KUKA KRL program: MyProgram_230().src

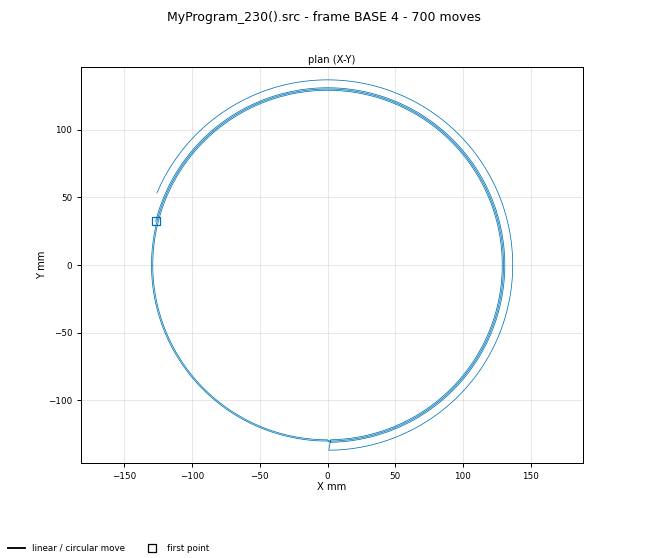
[picture p0: tool path of MyProgram_230().src in frame BASE 4, 700 of 700 moves have a stored position in this frame; points joined in program order, loops and branches not executed]
&ACCESS RVP
&REL 1
&PARAM TEMPLATE = C:\KRC\Roboter\Template\vorgabe
&PARAM EDITMASK = *
DEF MyProgram_230()
; ---- Setting reference (Base) ----
$BASE = BASE_DATA[4]

; --------------------------
; ---- Setting tool (TCP) ----
$TOOL = TOOL_DATA[3]
; --------------------------

$VEL.CP = VEL_APROX_PRINT
Startdeposition()
$VEL.CP = VEL_PRINT
LIN {X -126.9294,Y 32.2253,Z 157,A 163.8285,B 18.3414,C -0.4875,E1 18.1927,E2 284.7259} C_DIS
LIN {X -125.904,Y 36.0324,Z 157,A 161.9446,B 18.3414,C -0.4875,E1 18.1941,E2 286.6256} C_DIS
LIN {X -124.7405,Y 39.8661,Z 157,A 160.3345,B 18.3411,C -0.4975,E1 18.1954,E2 288.2164} C_DIS
LIN {X -123.6623,Y 43.0949,Z 157,A 158.8283,B 18.3411,C -0.5013,E1 18.1968,E2 289.7223} C_DIS
LIN {X -122.5468,Y 46.1718,Z 157,A 157.3766,B 18.3409,C -0.5049,E1 18.1982,E2 291.1743} C_DIS
LIN {X -121.4032,Y 49.0996,Z 157,A 155.9825,B 18.3409,C -0.5083,E1 18.1996,E2 292.5684} C_DIS
LIN {X -119.9916,Y 52.4573,Z 157,A 154.3901,B 18.3407,C -0.513,E1 18.2013,E2 294.1583} C_DIS
LIN {X -117.3041,Y 58.2179,Z 157,A 151.6663,B 18.3405,C -0.5228,E1 18.2046,E2 296.8714} C_DIS
LIN {X -116.1041,Y 60.5758,Z 157,A 149.9342,B 18.3409,C -0.5068,E1 18.2069,E2 298.6678} C_DIS
LIN {X -114.0894,Y 64.2932,Z 157,A 148.54,B 18.3403,C -0.5272,E1 18.2087,E2 300.007} C_DIS
LIN {X -112.0031,Y 67.8624,Z 157,A 146.6599,B 18.3403,C -0.5297,E1 18.2114,E2 301.8927} C_DIS
LIN {X -109.7276,Y 71.4835,Z 157,A 144.7555,B 18.3402,C -0.5336,E1 18.2143,E2 303.7982} C_DIS
LIN {X -107.2573,Y 75.1401,Z 157,A 142.8027,B 18.34,C -0.5379,E1 18.2174,E2 305.7508} C_DIS
LIN {X -104.7432,Y 78.6064,Z 157,A 140.9069,B 18.34,C -0.542,E1 18.2205,E2 307.6465} C_DIS
LIN {X -102.0917,Y 82.0203,Z 157,A 138.9861,B 18.3398,C -0.5458,E1 18.2238,E2 309.568} C_DIS
LIN {X -99.1429,Y 85.561,Z 157,A 136.9936,B 18.3396,C -0.5515,E1 18.2274,E2 311.5549} C_DIS
LIN {X -96.2928,Y 88.7565,Z 157,A 135.0913,B 18.3396,C -0.555,E1 18.231,E2 313.4579} C_DIS
LIN {X -93.2172,Y 91.982,Z 157,A 133.0947,B 18.3395,C -0.5579,E1 18.2349,E2 315.4573} C_DIS
LIN {X -90.087,Y 95.0495,Z 157,A 131.1811,B 18.3393,C -0.5624,E1 18.2387,E2 317.3678} C_DIS
LIN {X -86.7985,Y 98.0612,Z 157,A 129.232,B 18.3392,C -0.5667,E1 18.2428,E2 319.3141} C_DIS
LIN {X -83.2978,Y 101.0522,Z 157,A 127.211,B 18.3391,C -0.5707,E1 18.2471,E2 321.3333} C_DIS
LIN {X -79.8786,Y 103.7765,Z 157,A 125.2544,B 18.3391,C -0.573,E1 18.2514,E2 323.2926} C_DIS
LIN {X -76.3559,Y 106.3946,Z 157,A 123.3696,B 18.3389,C -0.5779,E1 18.2556,E2 325.1709} C_DIS
LIN {X -72.8799,Y 108.8051,Z 157,A 121.4838,B 18.3388,C -0.5802,E1 18.26,E2 327.0585} C_DIS
LIN {X -69.4414,Y 111.0314,Z 157,A 119.7018,B 18.3387,C -0.5837,E1 18.2642,E2 328.8372} C_DIS
LIN {X -65.8977,Y 113.1706,Z 157,A 117.8352,B 18.3387,C -0.5848,E1 18.2687,E2 330.7082} C_DIS
LIN {X -61.9917,Y 115.356,Z 157,A 115.6717,B 18.3387,C -0.5808,E1 18.274,E2 332.893} C_DIS
LIN {X -59.1213,Y 116.8514,Z 157,A 114.6066,B 18.3383,C -0.5952,E1 18.2766,E2 333.9162} C_DIS
LIN {X -56.0403,Y 118.3603,Z 157,A 112.9696,B 18.3384,C -0.5927,E1 18.2807,E2 335.5674} C_DIS
LIN {X -48.8655,Y 121.4976,Z 157,A 109.6259,B 18.3382,C -0.6001,E1 18.2893,E2 338.8981} C_DIS
LIN {X -45.691,Y 122.7269,Z 157,A 108.1493,B 18.3381,C -0.6024,E1 18.2931,E2 340.3718} C_DIS
LIN {X -42.2196,Y 123.9658,Z 157,A 106.4116,B 18.3381,C -0.5998,E1 18.2977,E2 342.1225} C_DIS
LIN {X -38.1423,Y 125.2785,Z 157,A 104.655,B 18.338,C -0.606,E1 18.3024,E2 343.8638} C_DIS
LIN {X -35.0335,Y 126.1834,Z 157,A 103.2075,B 18.338,C -0.6062,E1 18.3062,E2 345.3137} C_DIS
LIN {X -27.6513,Y 128.0037,Z 157,A 99.8455,B 18.338,C -0.6078,E1 18.3154,E2 348.6771} C_DIS
LIN {X -20.6201,Y 129.3241,Z 157,A 96.6623,B 18.338,C -0.6079,E1 18.3241,E2 351.8643} C_DIS
LIN {X -15.0154,Y 130.093,Z 157,A 94.0812,B 18.338,C -0.6054,E1 18.3313,E2 354.456} C_DIS
LIN {X -11.0032,Y 130.4934,Z 157,A 92.4941,B 18.3378,C -0.6126,E1 18.3357,E2 356.0216} C_DIS
LIN {X -6.9018,Y 130.7749,Z 157,A 90.6614,B 18.3378,C -0.6119,E1 18.3408,E2 357.8572} C_DIS
LIN {X -3.0947,Y 130.9211,Z 157,A 89.0121,B 18.3378,C -0.6129,E1 18.3454,E2 359.5036} C_DIS
LIN {X 0.7077,Y 130.9547,Z 157,A 87.3244,B 18.3378,C -0.6123,E1 18.3501,E2 361.1932} C_DIS
LIN {X 4.9525,Y 130.8629,Z 157,A 85.4948,B 18.3378,C -0.6134,E1 18.3552,E2 363.0188} C_DIS
LIN {X 8.8445,Y 130.6593,Z 157,A 83.69,B 18.3378,C -0.6096,E1 18.3603,E2 364.8345} C_DIS
LIN {X 12.681,Y 130.3411,Z 157,A 82.1185,B 18.3378,C -0.6135,E1 18.3646,E2 366.3922} C_DIS
LIN {X 16.8208,Y 129.8718,Z 157,A 80.0899,B 18.338,C -0.6055,E1 18.3703,E2 368.4441} C_DIS
LIN {X 21.4829,Y 129.1822,Z 157,A 78.2047,B 18.3378,C -0.6113,E1 18.3754,E2 370.3082} C_DIS
LIN {X 26.623,Y 128.2226,Z 157,A 75.8818,B 18.3378,C -0.6089,E1 18.3818,E2 372.6348} C_DIS
LIN {X 30.47,Y 127.3623,Z 157,A 74.2016,B 18.3378,C -0.6096,E1 18.3864,E2 374.3096} C_DIS
LIN {X 34.0088,Y 126.4635,Z 157,A 72.3281,B 18.3382,C -0.5982,E1 18.3915,E2 376.2149} C_DIS
LIN {X 37.1976,Y 125.5629,Z 157,A 71.2631,B 18.3378,C -0.6115,E1 18.3942,E2 377.2351} C_DIS
LIN {X 39.9846,Y 124.7027,Z 157,A 69.9298,B 18.3379,C -0.6084,E1 18.3978,E2 378.575} C_DIS
LIN {X 43.2512,Y 123.6082,Z 157,A 68.3028,B 18.3381,C -0.6025,E1 18.4021,E2 380.2161} C_DIS
LIN {X 47.2394,Y 122.1392,Z 157,A 66.5756,B 18.338,C -0.6057,E1 18.4066,E2 381.9279} C_DIS
LIN {X 50.5263,Y 120.8163,Z 157,A 64.9972,B 18.338,C -0.603,E1 18.4107,E2 383.5097} C_DIS
LIN {X 53.888,Y 119.3557,Z 157,A 63.2995,B 18.3383,C -0.5976,E1 18.4151,E2 385.2186} C_DIS
LIN {X 57.8507,Y 117.4852,Z 157,A 61.4569,B 18.3383,C -0.5981,E1 18.4197,E2 387.0529} C_DIS
LIN {X 60.9785,Y 115.8926,Z 157,A 59.9952,B 18.3383,C -0.599,E1 18.4233,E2 388.5062} C_DIS
LIN {X 64.5859,Y 113.9244,Z 157,A 58.0353,B 18.3385,C -0.5902,E1 18.4281,E2 390.4856} C_DIS
LIN {X 68.6354,Y 111.5312,Z 157,A 56.0373,B 18.3385,C -0.5895,E1 18.4329,E2 392.4773} C_DIS
LIN {X 72.3786,Y 109.1397,Z 157,A 54.0704,B 18.3386,C -0.5855,E1 18.4375,E2 394.4477} C_DIS
LIN {X 76.0983,Y 106.5788,Z 157,A 52.1676,B 18.3386,C -0.585,E1 18.4418,E2 396.3427} C_DIS
LIN {X 79.4898,Y 104.0738,Z 157,A 50.3093,B 18.3388,C -0.5813,E1 18.446,E2 398.2034} C_DIS
LIN {X 83.6518,Y 100.759,Z 157,A 47.9853,B 18.3388,C -0.5771,E1 18.451,E2 400.5282} C_DIS
LIN {X 87.0752,Y 97.8164,Z 157,A 45.6005,B 18.3395,C -0.5574,E1 18.4561,E2 402.962} C_DIS
LIN {X 90.2686,Y 94.877,Z 157,A 44.2587,B 18.3389,C -0.5752,E1 18.4587,E2 404.2399} C_DIS
LIN {X 92.9547,Y 92.2464,Z 157,A 42.5188,B 18.3392,C -0.5681,E1 18.4622,E2 405.992} C_DIS
LIN {X 96.4427,Y 88.5934,Z 157,A 40.3208,B 18.3392,C -0.5637,E1 18.4664,E2 408.1902} C_DIS
LIN {X 99.4064,Y 85.2551,Z 157,A 38.0738,B 18.3398,C -0.5478,E1 18.4706,E2 410.4732} C_DIS
LIN {X 101.7587,Y 82.4332,Z 157,A 36.8229,B 18.3395,C -0.5581,E1 18.4727,E2 411.6836} C_DIS
LIN {X 104.2925,Y 79.2036,Z 157,A 34.942,B 18.3397,C -0.5505,E1 18.4759,E2 413.5759} C_DIS
LIN {X 107.0744,Y 75.3993,Z 157,A 32.7589,B 18.34,C -0.5407,E1 18.4795,E2 415.775} C_DIS
LIN {X 109.5714,Y 71.7232,Z 157,A 31.0093,B 18.3399,C -0.5435,E1 18.4822,E2 417.5036} C_DIS
LIN {X 111.8857,Y 68.0565,Z 157,A 29.089,B 18.34,C -0.5377,E1 18.485,E2 419.4285} C_DIS
LIN {X 114.0229,Y 64.4115,Z 157,A 27.2622,B 18.3402,C -0.5338,E1 18.4876,E2 421.2545} C_DIS
LIN {X 116.1297,Y 60.5271,Z 157,A 25.4644,B 18.3402,C -0.534,E1 18.4899,E2 423.0383} C_DIS
LIN {X 118.128,Y 56.5266,Z 157,A 23.817,B 18.3399,C -0.5411,E1 18.4919,E2 424.6511} C_DIS
LIN {X 119.5942,Y 53.3548,Z 157,A 21.9933,B 18.3404,C -0.525,E1 18.4941,E2 426.5114} C_DIS
LIN {X 120.9373,Y 50.2366,Z 157,A 20.5149,B 18.3405,C -0.5211,E1 18.4957,E2 427.9907} C_DIS
LIN {X 122.3752,Y 46.63,Z 157,A 18.7053,B 18.3408,C -0.5119,E1 18.4975,E2 429.8154} C_DIS
LIN {X 123.6836,Y 43.0335,Z 157,A 17.1832,B 18.3408,C -0.5132,E1 18.4989,E2 431.3214} C_DIS
LIN {X 124.7092,Y 39.9644,Z 157,A 15.4546,B 18.3412,C -0.4966,E1 18.5005,E2 433.0887} C_DIS
LIN {X 125.6947,Y 36.7473,Z 157,A 14.3484,B 18.3409,C -0.5069,E1 18.5013,E2 434.1534} C_DIS
LIN {X 126.5682,Y 33.6161,Z 157,A 12.2036,B 18.3417,C -0.4738,E1 18.5029,E2 436.3852} C_DIS
LIN {X 127.8535,Y 28.347,Z 157,A 9.7574,B 18.342,C -0.4638,E1 18.5044,E2 438.8432} C_DIS
LIN {X 128.9712,Y 22.7181,Z 157,A 8.1043,B 18.3413,C -0.4905,E1 18.5052,E2 440.3984} C_DIS
LIN {X 129.573,Y 18.9896,Z 157,A 6.5375,B 18.3413,C -0.4889,E1 18.5059,E2 441.9573} C_DIS
LIN {X 129.8956,Y 16.6387,Z 157,A 5.2799,B 18.3417,C -0.4769,E1 18.5063,E2 443.2424} C_DIS
LIN {X 130.3759,Y 12.3184,Z 157,A 3.4277,B 18.3417,C -0.4731,E1 18.5069,E2 445.0912} C_DIS
LIN {X 130.7041,Y 8.1265,Z 157,A 1.6792,B 18.3418,C -0.4711,E1 18.5072,E2 446.8315} C_DIS
LIN {X 130.8872,Y 4.3132,Z 157,A -0.0996,B 18.342,C -0.4615,E1 18.5074,E2 448.6256} C_DIS
LIN {X 130.9598,Y -0.009,Z 157,A -1.9756,B 18.3422,C -0.4562,E1 18.5074,E2 450.5025} C_DIS
LIN {X 130.9012,Y -3.8099,Z 157,A -3.5163,B 18.3422,C -0.456,E1 18.5074,E2 452.031} C_DIS
LIN {X 130.7111,Y -8.0136,Z 157,A -5.3616,B 18.3423,C -0.4501,E1 18.5071,E2 453.8795} C_DIS
LIN {X 130.4586,Y -11.4149,Z 157,A -7.3892,B 18.3429,C -0.4239,E1 18.5066,E2 455.9728} C_DIS
LIN {X 129.9501,Y -16.2194,Z 157,A -8.8474,B 18.3425,C -0.4438,E1 18.5061,E2 457.3563} C_DIS
LIN {X 129.5124,Y -19.4037,Z 157,A -11.0028,B 18.3432,C -0.4093,E1 18.5052,E2 459.6027} C_DIS
LIN {X 128.6154,Y -24.6504,Z 157,A -12.2404,B 18.3424,C -0.4461,E1 18.5046,E2 460.714} C_DIS
LIN {X 127.9074,Y -28.0974,Z 157,A -14.1965,B 18.3429,C -0.4245,E1 18.5035,E2 462.7224} C_DIS
LIN {X 126.8202,Y -32.6552,Z 157,A -16.6656,B 18.3434,C -0.4013,E1 18.5018,E2 465.2444} C_DIS
LIN {X 125.6801,Y -36.7972,Z 157,A -18.0085,B 18.3431,C -0.4173,E1 18.5008,E2 466.5263} C_DIS
LIN {X 124.7062,Y -39.9737,Z 157,A -19.4412,B 18.3431,C -0.4137,E1 18.4996,E2 467.9587} C_DIS
LIN {X 123.6599,Y -43.1019,Z 157,A -20.9337,B 18.3433,C -0.4074,E1 18.4982,E2 469.4593} C_DIS
LIN {X 121.3565,Y -49.2155,Z 157,A -24.1781,B 18.3438,C -0.3835,E1 18.4949,E2 472.7539} C_DIS
LIN {X 119.7596,Y -52.9848,Z 157,A -25.3756,B 18.3434,C -0.4021,E1 18.4936,E2 473.8835} C_DIS
LIN {X 117.9672,Y -56.8625,Z 157,A -27.6334,B 18.3438,C -0.3811,E1 18.4909,E2 476.1905} C_DIS
LIN {X 115.717,Y -61.313,Z 157,A -29.5456,B 18.3438,C -0.3857,E1 18.4885,E2 478.0739} C_DIS
LIN {X 113.6109,Y -65.1355,Z 157,A -31.4921,B 18.3438,C -0.3789,E1 18.4858,E2 480.0277} C_DIS
LIN {X 111.4011,Y -68.8471,Z 157,A -33.4048,B 18.344,C -0.3728,E1 18.483,E2 481.9459} C_DIS
LIN {X 109.0509,Y -72.5117,Z 157,A -35.2937,B 18.344,C -0.3683,E1 18.4801,E2 483.8357} C_DIS
LIN {X 105.1496,Y -78.0614,Z 157,A -38.4139,B 18.3443,C -0.3544,E1 18.475,E2 486.9784} C_DIS
LIN {X 103.2003,Y -80.6213,Z 157,A -39.519,B 18.3442,C -0.3629,E1 18.4732,E2 488.0494} C_DIS
LIN {X 100.8196,Y -83.5786,Z 157,A -41.765,B 18.3447,C -0.3355,E1 18.4691,E2 490.3674} C_DIS
LIN {X 97.7182,Y -87.1845,Z 157,A -43.1658,B 18.3443,C -0.3574,E1 18.4666,E2 491.6901} C_DIS
LIN {X 93.7761,Y -91.4122,Z 157,A -45.7303,B 18.3444,C -0.35,E1 18.4617,E2 494.2624} C_DIS
LIN {X 88.8238,Y -96.2309,Z 157,A -48.6791,B 18.3445,C -0.346,E1 18.4558,E2 497.2064} C_DIS
LIN {X 85.7578,Y -98.9734,Z 157,A -50.5189,B 18.3446,C -0.3405,E1 18.4519,E2 499.0535} C_DIS
LIN {X 82.9407,Y -101.3451,Z 157,A -52.6039,B 18.345,C -0.3184,E1 18.4473,E2 501.1971} C_DIS
LIN {X 79.7464,Y -103.8776,Z 157,A -54.0484,B 18.3448,C -0.3281,E1 18.4442,E2 502.6035} C_DIS
LIN {X 76.0879,Y -106.5863,Z 157,A -55.914,B 18.3448,C -0.3292,E1 18.44,E2 504.4565} C_DIS
LIN {X 72.8224,Y -108.8435,Z 157,A -57.7068,B 18.3448,C -0.3237,E1 18.4359,E2 506.2581} C_DIS
LIN {X 67.2837,Y -112.352,Z 157,A -60.5464,B 18.345,C -0.3197,E1 18.4291,E2 509.0977} C_DIS
LIN {X 63.6471,Y -114.4513,Z 157,A -62.4076,B 18.345,C -0.3156,E1 18.4246,E2 510.9638} C_DIS
LIN {X 60.2839,Y -116.2574,Z 157,A -64.6109,B 18.3454,C -0.2923,E1 18.419,E2 513.2323} C_DIS
LIN {X 55.8016,Y -118.4744,Z 157,A -66.1122,B 18.345,C -0.3156,E1 18.4154,E2 514.6543} C_DIS
LIN {X 53.3864,Y -119.58,Z 157,A -67.302,B 18.345,C -0.3129,E1 18.4123,E2 515.8486} C_DIS
LIN {X 50.0023,Y -121.0352,Z 157,A -68.8725,B 18.345,C -0.3122,E1 18.4083,E2 517.4159} C_DIS
LIN {X 47.2558,Y -122.1328,Z 157,A -70.1866,B 18.3451,C -0.3098,E1 18.4049,E2 518.7336} C_DIS
LIN {X 43.8983,Y -123.3805,Z 157,A -71.7434,B 18.3451,C -0.3082,E1 18.4008,E2 520.2907} C_DIS
LIN {X 40.3453,Y -124.5875,Z 157,A -73.8583,B 18.3455,C -0.2882,E1 18.395,E2 522.4634} C_DIS
LIN {X 36.5141,Y -125.763,Z 157,A -74.7263,B 18.345,C -0.3204,E1 18.393,E2 523.2272} C_DIS
LIN {X 31.9984,Y -126.987,Z 157,A -77.0681,B 18.3452,C -0.307,E1 18.3866,E2 525.6063} C_DIS
LIN {X 24.0037,Y -128.739,Z 157,A -80.4298,B 18.3451,C -0.3123,E1 18.3775,E2 528.9448} C_DIS
LIN {X 20.8342,Y -129.2893,Z 157,A -82.0846,B 18.3453,C -0.3019,E1 18.3728,E2 530.6303} C_DIS
LIN {X 18.5339,Y -129.6382,Z 157,A -83.1745,B 18.3453,C -0.2985,E1 18.3698,E2 531.7295} C_DIS
LIN {X 14.887,Y -130.109,Z 157,A -84.9132,B 18.3453,C -0.2927,E1 18.3649,E2 533.4848} C_DIS
LIN {X 10.8445,Y -130.5068,Z 157,A -86.564,B 18.3453,C -0.2966,E1 18.3604,E2 535.1216} C_DIS
LIN {X 6.7871,Y -130.7807,Z 157,A -88.3914,B 18.3453,C -0.2942,E1 18.3553,E2 536.9558} C_DIS
LIN {X 2.4911,Y -130.9332,Z 157,A -90.297,B 18.3453,C -0.2927,E1 18.3499,E2 538.8653} C_DIS
LIN {X 2.4911,Y -130.9332,Z 157,A -90.297,B 18.3453,C -0.2927,E1 18.3499,E2 538.8653} C_DIS
Enddeposition()
LIN {X 0.9057,Y -130.0191,Z 157,A -89.6003,B 15.4645,C -0.0312,E1 15.4666,E2 538.886} C_DIS
Startdeposition()
$VEL.CP = VEL_PRINT
LIN {X 4.0156,Y -129.9636,Z 157,A -87.956,B 15.4645,C -0.0402,E1 15.4713,E2 537.2085} C_DIS
LIN {X 7.9,Y -129.7848,Z 157,A -86.3512,B 15.4645,C -0.0372,E1 15.4758,E2 535.6157} C_DIS
LIN {X 11.0255,Y -129.5567,Z 157,A -84.83,B 15.4645,C -0.0423,E1 15.48,E2 534.0769} C_DIS
LIN {X 14.969,Y -129.1611,Z 157,A -83.114,B 15.4645,C -0.0422,E1 15.4848,E2 532.3635} C_DIS
LIN {X 19.266,Y -128.5912,Z 157,A -80.8099,B 15.4645,C -0.0561,E1 15.4913,E2 530.0108} C_DIS
LIN {X 23.11,Y -127.9548,Z 157,A -79.687,B 15.4645,C -0.0379,E1 15.4942,E2 528.958} C_DIS
LIN {X 27.0142,Y -127.1883,Z 157,A -77.3504,B 15.4645,C -0.0583,E1 15.5008,E2 526.5501} C_DIS
LIN {X 30.8925,Y -126.3023,Z 157,A -76.0012,B 15.4645,C -0.0465,E1 15.5043,E2 525.2482} C_DIS
LIN {X 34.8635,Y -125.2637,Z 157,A -74.0967,B 15.4645,C -0.0514,E1 15.5095,E2 523.3308} C_DIS
LIN {X 42.0286,Y -123.0461,Z 157,A -70.951,B 15.4645,C -0.0497,E1 15.5178,E2 520.2014} C_DIS
LIN {X 44.8514,Y -122.0466,Z 157,A -69.4939,B 15.4645,C -0.0557,E1 15.5217,E2 518.7268} C_DIS
LIN {X 48.5461,Y -120.622,Z 157,A -67.9155,B 15.4645,C -0.0525,E1 15.5257,E2 517.1666} C_DIS
LIN {X 53.4488,Y -118.5317,Z 157,A -65.6314,B 15.4645,C -0.0535,E1 15.5316,E2 514.8881} C_DIS
LIN {X 59.8994,Y -115.4071,Z 157,A -62.0071,B 15.4644,C -0.0737,E1 15.5408,E2 511.2047} C_DIS
LIN {X 63.3148,Y -113.5705,Z 157,A -60.6306,B 15.4644,C -0.0653,E1 15.5441,E2 509.8665} C_DIS
LIN {X 67.0418,Y -111.4108,Z 157,A -58.5868,B 15.4644,C -0.0733,E1 15.549,E2 507.8032} C_DIS
LIN {X 71.371,Y -108.688,Z 157,A -56.5267,B 15.4644,C -0.0708,E1 15.5538,E2 505.7639} C_DIS
LIN {X 74.8406,Y -106.3286,Z 157,A -54.6933,B 15.4644,C -0.0737,E1 15.558,E2 503.9303} C_DIS
LIN {X 78.2629,Y -103.8355,Z 157,A -52.8336,B 15.4644,C -0.0771,E1 15.5622,E2 502.0692} C_DIS
LIN {X 81.8081,Y -101.0661,Z 157,A -50.8553,B 15.4644,C -0.0809,E1 15.5665,E2 500.0891} C_DIS
LIN {X 84.9845,Y -98.41,Z 157,A -49.0772,B 15.4644,C -0.0831,E1 15.5703,E2 498.3144} C_DIS
LIN {X 87.8139,Y -95.894,Z 157,A -47.3554,B 15.4643,C -0.0885,E1 15.5739,E2 496.5841} C_DIS
LIN {X 91.5561,Y -92.3276,Z 157,A -45.144,B 15.4643,C -0.0913,E1 15.5783,E2 494.378} C_DIS
LIN {X 94.3898,Y -89.4289,Z 157,A -43.3243,B 15.4643,C -0.0965,E1 15.5818,E2 492.5521} C_DIS
LIN {X 98.0775,Y -85.3679,Z 157,A -40.8126,B 15.4642,C -0.1055,E1 15.5865,E2 490.0259} C_DIS
LIN {X 101.2937,Y -81.5259,Z 157,A -38.7637,B 15.4642,C -0.1055,E1 15.5901,E2 487.9933} C_DIS
LIN {X 103.737,Y -78.3934,Z 157,A -37.2458,B 15.4642,C -0.1018,E1 15.5927,E2 486.5009} C_DIS
LIN {X 105.3421,Y -76.2229,Z 157,A -35.7451,B 15.4642,C -0.1155,E1 15.5952,E2 484.9615} C_DIS
LIN {X 108.0415,Y -72.346,Z 157,A -33.8505,B 15.4642,C -0.1144,E1 15.5981,E2 483.0865} C_DIS
LIN {X 110.1165,Y -69.1471,Z 157,A -32.1214,B 15.4641,C -0.1205,E1 15.6008,E2 481.3494} C_DIS
LIN {X 112.3499,Y -65.4562,Z 157,A -30.2335,B 15.4641,C -0.1252,E1 15.6034,E2 479.4605} C_DIS
LIN {X 114.3981,Y -61.8065,Z 157,A -28.3853,B 15.4641,C -0.1303,E1 15.6059,E2 477.6094} C_DIS
LIN {X 116.1477,Y -58.4503,Z 157,A -26.3714,B 15.4639,C -0.147,E1 15.6085,E2 475.5515} C_DIS
LIN {X 117.8855,Y -54.8588,Z 157,A -25.0697,B 15.4639,C -0.136,E1 15.61,E2 474.3023} C_DIS
LIN {X 119.338,Y -51.6219,Z 157,A -23.7477,B 15.4639,C -0.1321,E1 15.6115,E2 473.007} C_DIS
LIN {X 122.2827,Y -44.1966,Z 157,A -20.0067,B 15.4639,C -0.1498,E1 15.6153,E2 469.2351} C_DIS
LIN {X 123.6436,Y -40.239,Z 157,A -18.1651,B 15.4638,C -0.1551,E1 15.6169,E2 467.3914} C_DIS
LIN {X 124.6271,Y -37.0784,Z 157,A -16.8422,B 15.4638,C -0.1547,E1 15.618,E2 466.0828} C_DIS
LIN {X 125.554,Y -33.8039,Z 157,A -15.2352,B 15.4638,C -0.1628,E1 15.6192,E2 464.4609} C_DIS
LIN {X 126.4634,Y -30.2243,Z 157,A -13.6731,B 15.4637,C -0.1654,E1 15.6203,E2 462.9044} C_DIS
LIN {X 127.032,Y -27.7381,Z 157,A -12.2828,B 15.4635,C -0.178,E1 15.6211,E2 461.4808} C_DIS
LIN {X 127.9612,Y -23.0743,Z 157,A -10.4939,B 15.4635,C -0.1737,E1 15.622,E2 459.7257} C_DIS
LIN {X 128.7961,Y -17.8421,Z 157,A -8.1167,B 15.4635,C -0.1821,E1 15.623,E2 457.3405} C_DIS
LIN {X 129.5447,Y -11.1678,Z 157,A -4.857,B 15.4633,C -0.2016,E1 15.6239,E2 454.0411} C_DIS
LIN {X 129.8205,Y -7.3209,Z 157,A -3.4619,B 15.4633,C -0.1961,E1 15.6242,E2 452.6803} C_DIS
LIN {X 129.9807,Y -3.4033,Z 157,A -1.8356,B 15.4633,C -0.1978,E1 15.6243,E2 451.0638} C_DIS
LIN {X 130.0252,Y 0.5219,Z 157,A -0.0574,B 15.4633,C -0.2047,E1 15.6243,E2 449.2776} C_DIS
LIN {X 129.9329,Y 4.8962,Z 157,A 1.8011,B 15.4632,C -0.2081,E1 15.6242,E2 447.425} C_DIS
LIN {X 129.7017,Y 9.1675,Z 157,A 3.6535,B 15.4632,C -0.2127,E1 15.6239,E2 445.5741} C_DIS
LIN {X 129.447,Y 12.2466,Z 157,A 4.9885,B 15.4631,C -0.2159,E1 15.6235,E2 444.2406} C_DIS
LIN {X 129.0375,Y 16.005,Z 157,A 6.5847,B 15.4631,C -0.2184,E1 15.623,E2 442.6507} C_DIS
LIN {X 128.1711,Y 21.8832,Z 157,A 8.9753,B 15.4631,C -0.2184,E1 15.622,E2 440.2841} C_DIS
LIN {X 127.1017,Y 27.4155,Z 157,A 11.8677,B 15.4627,C -0.2398,E1 15.6204,E2 437.3405} C_DIS
LIN {X 125.8049,Y 32.8631,Z 157,A 14.1393,B 15.4627,C -0.2402,E1 15.6189,E2 435.0894} C_DIS
LIN {X 124.8575,Y 36.2916,Z 157,A 15.7154,B 15.4627,C -0.245,E1 15.6177,E2 433.5106} C_DIS
LIN {X 123.5487,Y 40.5272,Z 157,A 17.6736,B 15.4626,C -0.2507,E1 15.616,E2 431.5498} C_DIS
LIN {X 122.4074,Y 43.8508,Z 157,A 19.137,B 15.4626,C -0.2522,E1 15.6147,E2 430.0949} C_DIS
LIN {X 121.3399,Y 46.7247,Z 157,A 20.4392,B 15.4625,C -0.2543,E1 15.6134,E2 428.7971} C_DIS
LIN {X 120.2128,Y 49.5542,Z 157,A 21.791,B 15.4625,C -0.2583,E1 15.612,E2 427.4429} C_DIS
LIN {X 118.8229,Y 52.7976,Z 157,A 23.2778,B 15.4625,C -0.2602,E1 15.6103,E2 425.9626} C_DIS
LIN {X 117.6508,Y 55.3624,Z 157,A 25.1018,B 15.462,C -0.2835,E1 15.6081,E2 424.0685} C_DIS
LIN {X 115.7449,Y 59.2415,Z 157,A 26.4719,B 15.4622,C -0.2702,E1 15.6064,E2 422.7601} C_DIS
LIN {X 113.9197,Y 62.6841,Z 157,A 28.2009,B 15.4622,C -0.2751,E1 15.6041,E2 421.0283} C_DIS
LIN {X 111.9602,Y 66.1202,Z 157,A 29.9007,B 15.4621,C -0.2781,E1 15.6017,E2 419.3321} C_DIS
LIN {X 109.8139,Y 69.6266,Z 157,A 31.6839,B 15.4621,C -0.2817,E1 15.5991,E2 417.5507} C_DIS
LIN {X 108.1191,Y 72.2297,Z 157,A 33.695,B 15.4616,C -0.3069,E1 15.5959,E2 415.4625} C_DIS
LIN {X 105.2646,Y 76.3298,Z 157,A 35.2887,B 15.4619,C -0.2915,E1 15.5934,E2 413.9393} C_DIS
LIN {X 102.6551,Y 79.805,Z 157,A 37.2157,B 15.4618,C -0.2964,E1 15.5901,E2 412.0094} C_DIS
LIN {X 100.6184,Y 82.3579,Z 157,A 38.7099,B 15.4617,C -0.3015,E1 15.5875,E2 410.5078} C_DIS
LIN {X 97.7034,Y 85.7968,Z 157,A 40.6571,B 15.4617,C -0.3046,E1 15.5839,E2 408.564} C_DIS
LIN {X 94.9386,Y 88.8462,Z 157,A 42.2931,B 15.4617,C -0.3025,E1 15.5809,E2 406.9478} C_DIS
LIN {X 92.4744,Y 91.4083,Z 157,A 44.0155,B 15.4615,C -0.311,E1 15.5775,E2 405.2062} C_DIS
LIN {X 89.3563,Y 94.4583,Z 157,A 45.9962,B 15.4614,C -0.3168,E1 15.5735,E2 403.2175} C_DIS
LIN {X 85.7235,Y 97.7673,Z 157,A 48.0629,B 15.4614,C -0.3177,E1 15.5692,E2 401.1615} C_DIS
LIN {X 82.2979,Y 100.6674,Z 157,A 50.0289,B 15.4613,C -0.321,E1 15.565,E2 399.196} C_DIS
LIN {X 78.7142,Y 103.4943,Z 157,A 52.0385,B 15.4613,C -0.3245,E1 15.5605,E2 397.1858} C_DIS
LIN {X 75.2987,Y 106.0054,Z 157,A 53.8661,B 15.4612,C -0.3263,E1 15.5564,E2 395.3623} C_DIS
LIN {X 71.9451,Y 108.3091,Z 157,A 55.6844,B 15.4612,C -0.33,E1 15.5522,E2 393.5405} C_DIS
LIN {X 68.2098,Y 110.6994,Z 157,A 57.4518,B 15.4612,C -0.3269,E1 15.548,E2 391.7944} C_DIS
LIN {X 64.7919,Y 112.7344,Z 157,A 59.3602,B 15.461,C -0.3345,E1 15.5434,E2 389.8675} C_DIS
LIN {X 61.3831,Y 114.6256,Z 157,A 61.0614,B 15.461,C -0.3363,E1 15.5392,E2 388.1678} C_DIS
LIN {X 57.6238,Y 116.5585,Z 157,A 62.7386,B 15.461,C -0.3326,E1 15.5351,E2 386.512} C_DIS
LIN {X 54.4923,Y 118.0549,Z 157,A 64.3177,B 15.461,C -0.3361,E1 15.5311,E2 384.9269} C_DIS
LIN {X 51.5211,Y 119.3816,Z 157,A 65.6649,B 15.461,C -0.3349,E1 15.5277,E2 383.5897} C_DIS
LIN {X 47.8458,Y 120.9041,Z 157,A 67.5866,B 15.4608,C -0.3421,E1 15.5227,E2 381.6484} C_DIS
LIN {X 44.2051,Y 122.2797,Z 157,A 69.2161,B 15.4608,C -0.3411,E1 15.5184,E2 380.0289} C_DIS
LIN {X 41.3088,Y 123.2885,Z 157,A 70.6148,B 15.4608,C -0.3437,E1 15.5147,E2 378.6247} C_DIS
LIN {X 37.5075,Y 124.4987,Z 157,A 72.4986,B 15.4607,C -0.3492,E1 15.5096,E2 376.7264} C_DIS
LIN {X 33.6761,Y 125.5881,Z 157,A 74.0966,B 15.4607,C -0.3454,E1 15.5054,E2 375.1469} C_DIS
LIN {X 29.7879,Y 126.5686,Z 157,A 75.9567,B 15.4607,C -0.3494,E1 15.5003,E2 373.2764} C_DIS
LIN {X 26.3708,Y 127.3233,Z 157,A 77.3448,B 15.4607,C -0.3454,E1 15.4966,E2 371.9064} C_DIS
LIN {X 23.7925,Y 127.831,Z 157,A 78.8582,B 15.4605,C -0.3571,E1 15.4923,E2 370.3519} C_DIS
LIN {X 20.4863,Y 128.4022,Z 157,A 79.9077,B 15.4608,C -0.3442,E1 15.4896,E2 369.3527} C_DIS
LIN {X 14.2539,Y 129.2417,Z 157,A 82.8254,B 15.4607,C -0.3495,E1 15.4814,E2 366.419} C_DIS
LIN {X 10.4865,Y 129.6022,Z 157,A 84.5649,B 15.4607,C -0.3521,E1 15.4766,E2 364.6718} C_DIS
LIN {X 6.4419,Y 129.8654,Z 157,A 86.2491,B 15.4607,C -0.349,E1 15.4719,E2 363.0001} C_DIS
LIN {X 2.7918,Y 129.9966,Z 157,A 87.9619,B 15.4607,C -0.3522,E1 15.4671,E2 361.2761} C_DIS
LIN {X -1.2477,Y 130.0202,Z 157,A 89.7261,B 15.4607,C -0.3515,E1 15.4622,E2 359.5146} C_DIS
LIN {X -5.7874,Y 129.8982,Z 157,A 91.7277,B 15.4607,C -0.3511,E1 15.4566,E2 357.514} C_DIS
LIN {X -9.9002,Y 129.6483,Z 157,A 93.4428,B 15.4607,C -0.3475,E1 15.4518,E2 355.8115} C_DIS
LIN {X -12.5253,Y 129.4203,Z 157,A 95.5538,B 15.4601,C -0.3763,E1 15.4457,E2 353.5904} C_DIS
LIN {X -19.0643,Y 128.6214,Z 157,A 97.6322,B 15.4607,C -0.3494,E1 15.4402,E2 351.6103} C_DIS
LIN {X -27.4806,Y 127.0876,Z 157,A 101.2856,B 15.4608,C -0.3433,E1 15.4302,E2 347.9732} C_DIS
LIN {X -32.577,Y 125.8791,Z 157,A 103.7474,B 15.4608,C -0.3461,E1 15.4235,E2 345.4954} C_DIS
LIN {X -36.9689,Y 124.6592,Z 157,A 105.7099,B 15.4608,C -0.3428,E1 15.4183,E2 343.5398} C_DIS
LIN {X -40.6992,Y 123.4914,Z 157,A 107.526,B 15.4608,C -0.3438,E1 15.4134,E2 341.7143} C_DIS
LIN {X -45.2409,Y 121.9008,Z 157,A 109.4604,B 15.461,C -0.3359,E1 15.4084,E2 339.8033} C_DIS
LIN {X -48.3115,Y 120.7166,Z 157,A 110.7218,B 15.4611,C -0.3286,E1 15.4052,E2 338.5649} C_DIS
LIN {X -52.3514,Y 119.0225,Z 157,A 112.9245,B 15.4611,C -0.3341,E1 15.3994,E2 336.3328} C_DIS
LIN {X -55.6176,Y 117.5299,Z 157,A 114.4853,B 15.4611,C -0.3314,E1 15.3955,E2 334.7759} C_DIS
LIN {X -58.8496,Y 115.9444,Z 157,A 116.0499,B 15.4611,C -0.3284,E1 15.3916,E2 333.2153} C_DIS
LIN {X -62.0127,Y 114.2864,Z 157,A 117.8976,B 15.4611,C -0.3341,E1 15.387,E2 331.3376} C_DIS
LIN {X -66.525,Y 111.7198,Z 157,A 119.9727,B 15.4612,C -0.3242,E1 15.382,E2 329.2895} C_DIS
LIN {X -69.7761,Y 109.7193,Z 157,A 121.7423,B 15.4612,C -0.3239,E1 15.3778,E2 327.5116} C_DIS
LIN {X -73.4153,Y 107.3178,Z 157,A 123.6604,B 15.4612,C -0.3204,E1 15.3734,E2 325.596} C_DIS
LIN {X -77.0706,Y 104.7235,Z 157,A 125.5962,B 15.4614,C -0.3156,E1 15.369,E2 323.667} C_DIS
LIN {X -80.5094,Y 102.1037,Z 157,A 127.5676,B 15.4614,C -0.3138,E1 15.3646,E2 321.69} C_DIS
LIN {X -83.7825,Y 99.4356,Z 157,A 129.3903,B 15.4615,C -0.309,E1 15.3607,E2 319.8739} C_DIS
LIN {X -86.9195,Y 96.7053,Z 157,A 131.2681,B 15.4615,C -0.3065,E1 15.3568,E2 317.993} C_DIS
LIN {X -90.1455,Y 93.7061,Z 157,A 133.2477,B 15.4616,C -0.3034,E1 15.3528,E2 316.0114} C_DIS
LIN {X -93.2224,Y 90.6451,Z 157,A 135.1885,B 15.4616,C -0.3,E1 15.349,E2 314.0697} C_DIS
LIN {X -96.2992,Y 87.369,Z 157,A 137.1461,B 15.4618,C -0.2948,E1 15.3453,E2 312.1172} C_DIS
LIN {X -99.2634,Y 83.9866,Z 157,A 139.1491,B 15.4618,C -0.2907,E1 15.3416,E2 310.1142} C_DIS
LIN {X -101.8689,Y 80.8063,Z 157,A 140.9397,B 15.462,C -0.2857,E1 15.3385,E2 308.3284} C_DIS
LIN {X -104.3293,Y 77.6033,Z 157,A 142.7498,B 15.462,C -0.2822,E1 15.3355,E2 306.517} C_DIS
LIN {X -106.9024,Y 74.0192,Z 157,A 144.7437,B 15.462,C -0.2786,E1 15.3322,E2 304.5199} C_DIS
LIN {X -109.3187,Y 70.4019,Z 157,A 146.6757,B 15.4622,C -0.2741,E1 15.3293,E2 302.5887} C_DIS
LIN {X -111.6226,Y 66.688,Z 157,A 148.6676,B 15.4622,C -0.2709,E1 15.3264,E2 300.5916} C_DIS
LIN {X -113.8627,Y 62.7869,Z 157,A 151.0426,B 15.4622,C -0.2767,E1 15.3231,E2 298.1736} C_DIS
LIN {X -115.8287,Y 59.0769,Z 157,A 152.7247,B 15.4622,C -0.2669,E1 15.321,E2 296.5135} C_DIS
LIN {X -117.3328,Y 56.0302,Z 157,A 153.9997,B 15.4625,C -0.2564,E1 15.3195,E2 295.2663} C_DIS
LIN {X -119.3211,Y 51.6609,Z 157,A 156.0904,B 15.4625,C -0.2498,E1 15.3171,E2 293.1813} C_DIS
LIN {X -120.9212,Y 47.801,Z 157,A 158.008,B 15.4626,C -0.2467,E1 15.3151,E2 291.2574} C_DIS
LIN {X -122.2324,Y 44.3361,Z 157,A 159.5349,B 15.4627,C -0.239,E1 15.3136,E2 289.7449} C_DIS
LIN {X -123.3078,Y 41.2508,Z 157,A 161.0048,B 15.4627,C -0.2357,E1 15.3123,E2 288.2735} C_DIS
LIN {X -124.3673,Y 37.9366,Z 157,A 162.5484,B 15.4628,C -0.2315,E1 15.311,E2 286.7307} C_DIS
LIN {X -125.4574,Y 34.1664,Z 157,A 164.4173,B 15.4628,C -0.2303,E1 15.3096,E2 284.8479} C_DIS
LIN {X -126.4214,Y 30.3985,Z 157,A 166.0393,B 15.463,C -0.2227,E1 15.3085,E2 283.2388} C_DIS
LIN {X -127.2876,Y 26.5463,Z 157,A 167.886,B 15.463,C -0.2205,E1 15.3074,E2 281.3821} C_DIS
LIN {X -128.1583,Y 21.9595,Z 157,A 169.9284,B 15.463,C -0.2139,E1 15.3064,E2 279.3441} C_DIS
LIN {X -128.7043,Y 18.4843,Z 157,A 171.4583,B 15.4632,C -0.2087,E1 15.3058,E2 277.8185} C_DIS
LIN {X -129.2412,Y 14.2591,Z 157,A 173.2908,B 15.4632,C -0.2018,E1 15.3052,E2 275.9937} C_DIS
LIN {X -129.5055,Y 11.6313,Z 157,A 174.4518,B 15.4632,C -0.1982,E1 15.3049,E2 274.8346} C_DIS
LIN {X -129.8334,Y 7.0768,Z 157,A 176.5627,B 15.4633,C -0.1948,E1 15.3045,E2 272.7148} C_DIS
LIN {X -130.0216,Y 1.0585,Z 157,A 179.8048,B 15.4633,C -0.2034,E1 15.3043,E2 269.4072} C_DIS
LIN {X -129.9757,Y -3.5833,Z 157,A -178.7143,B 15.4635,C -0.1813,E1 15.3044,E2 267.9949} C_DIS
LIN {X -129.8208,Y -7.3163,Z 157,A -176.9934,B 15.4635,C -0.1784,E1 15.3047,E2 266.2674} C_DIS
LIN {X -129.3637,Y -13.1147,Z 157,A -174.3855,B 15.4636,C -0.172,E1 15.3053,E2 263.6575} C_DIS
LIN {X -129.0379,Y -16.0022,Z 157,A -172.9956,B 15.4636,C -0.1712,E1 15.3058,E2 262.2563} C_DIS
LIN {X -128.387,Y -20.5844,Z 157,A -171.0427,B 15.4637,C -0.1627,E1 15.3066,E2 260.3159} C_DIS
LIN {X -127.6474,Y -24.753,Z 157,A -169.2664,B 15.4637,C -0.1547,E1 15.3075,E2 258.5521} C_DIS
LIN {X -126.8401,Y -28.6032,Z 157,A -167.4601,B 15.4638,C -0.1517,E1 15.3086,E2 256.7393} C_DIS
LIN {X -126.0906,Y -31.7433,Z 157,A -166.0751,B 15.4638,C -0.1465,E1 15.3095,E2 255.3602} C_DIS
LIN {X -125.2856,Y -34.7851,Z 157,A -164.6435,B 15.4638,C -0.1438,E1 15.3105,E2 253.9249} C_DIS
LIN {X -124.3741,Y -37.9145,Z 157,A -163.1983,B 15.4639,C -0.1399,E1 15.3117,E2 252.4801} C_DIS
LIN {X -123.3438,Y -41.1427,Z 157,A -161.6618,B 15.4639,C -0.1369,E1 15.313,E2 250.9402} C_DIS
LIN {X -121.5054,Y -46.2966,Z 157,A -159.1544,B 15.4639,C -0.1329,E1 15.3154,E2 248.424} C_DIS
LIN {X -120.0741,Y -49.8863,Z 157,A -157.5804,B 15.464,C -0.1246,E1 15.3171,E2 246.8668} C_DIS
LIN {X -118.8361,Y -52.7682,Z 157,A -156.0902,B 15.464,C -0.1239,E1 15.3188,E2 245.3652} C_DIS
LIN {X -116.2496,Y -58.25,Z 157,A -153.2691,B 15.464,C -0.121,E1 15.3222,E2 242.529} C_DIS
LIN {X -114.285,Y -62.0153,Z 157,A -151.4375,B 15.4641,C -0.115,E1 15.3246,E2 240.7038} C_DIS
LIN {X -111.7286,Y -66.5102,Z 157,A -149.1812,B 15.4641,C -0.1086,E1 15.3278,E2 238.452} C_DIS
LIN {X -109.5225,Y -70.0835,Z 157,A -147.3492,B 15.4641,C -0.1035,E1 15.3305,E2 236.6237} C_DIS
LIN {X -106.5458,Y -74.5317,Z 157,A -144.9048,B 15.4642,C -0.1002,E1 15.3343,E2 234.1711} C_DIS
LIN {X -103.9544,Y -78.1053,Z 157,A -142.9401,B 15.4642,C -0.0962,E1 15.3376,E2 232.2055} C_DIS
LIN {X -101.7802,Y -80.9176,Z 157,A -141.1733,B 15.4642,C -0.0985,E1 15.3407,E2 230.4161} C_DIS
LIN {X -99.7329,Y -83.4281,Z 157,A -139.9393,B 15.4642,C -0.0897,E1 15.3429,E2 229.2058} C_DIS
LIN {X -96.8651,Y -86.7411,Z 157,A -138.0349,B 15.4643,C -0.0847,E1 15.3464,E2 227.3057} C_DIS
LIN {X -93.9393,Y -89.9015,Z 157,A -136.291,B 15.4643,C -0.0762,E1 15.3497,E2 225.5811} C_DIS
LIN {X -91.2731,Y -92.6078,Z 157,A -134.4158,B 15.4643,C -0.0787,E1 15.3534,E2 223.6831} C_DIS
LIN {X -88.4414,Y -95.3155,Z 157,A -132.6892,B 15.4643,C -0.0753,E1 15.3569,E2 221.9574} C_DIS
LIN {X -85.1827,Y -98.2393,Z 157,A -130.6874,B 15.4643,C -0.0738,E1 15.3611,E2 219.9479} C_DIS
LIN {X -81.8479,Y -101.034,Z 157,A -128.7622,B 15.4643,C -0.0706,E1 15.3653,E2 218.0226} C_DIS
LIN {X -78.2664,Y -103.8328,Z 157,A -126.8146,B 15.4644,C -0.0655,E1 15.3696,E2 216.0823} C_DIS
LIN {X -74.7005,Y -106.4275,Z 157,A -125.088,B 15.4644,C -0.0558,E1 15.3734,E2 214.382} C_DIS
LIN {X -71.2155,Y -108.7904,Z 157,A -122.1235,B 15.4644,C -0.0864,E1 15.3807,E2 211.286} C_DIS
LIN {X -65.7926,Y -112.1527,Z 157,A -120.197,B 15.4644,C -0.0555,E1 15.385,E2 209.4659} C_DIS
LIN {X -62.241,Y -114.1619,Z 157,A -118.3489,B 15.4644,C -0.0546,E1 15.3895,E2 207.6122} C_DIS
LIN {X -59.0627,Y -115.8359,Z 157,A -116.938,B 15.4644,C -0.0475,E1 15.393,E2 206.2219} C_DIS
LIN {X -56.7353,Y -116.9959,Z 157,A -115.556,B 15.4644,C -0.0532,E1 15.3965,E2 204.8121} C_DIS
LIN {X -53.4767,Y -118.5192,Z 157,A -114.1005,B 15.4644,C -0.0475,E1 15.4002,E2 203.3721} C_DIS
LIN {X -46.1576,Y -121.5575,Z 157,A -110.493,B 15.4644,C -0.0475,E1 15.4096,E2 199.7511} C_DIS
LIN {X -42.6907,Y -122.8166,Z 157,A -108.9344,B 15.4644,C -0.0441,E1 15.4136,E2 198.2003} C_DIS
LIN {X -39.6259,Y -123.8394,Z 157,A -107.4472,B 15.4644,C -0.0449,E1 15.4176,E2 196.7055} C_DIS
LIN {X -35.3744,Y -125.1208,Z 157,A -105.4705,B 15.4644,C -0.0442,E1 15.4229,E2 194.7261} C_DIS
LIN {X -31.5611,Y -126.1369,Z 157,A -103.803,B 15.4644,C -0.0409,E1 15.4274,E2 193.067} C_DIS
LIN {X -28.2035,Y -126.9314,Z 157,A -102.3317,B 15.4644,C -0.0386,E1 15.4314,E2 191.6013} C_DIS
LIN {X -24.4052,Y -127.7139,Z 157,A -100.5958,B 15.4644,C -0.0386,E1 15.4361,E2 189.8617} C_DIS
LIN {X -21.5211,Y -128.2315,Z 157,A -98.7046,B 15.4644,C -0.0571,E1 15.4416,E2 187.8983} C_DIS
LIN {X -16.868,Y -128.9261,Z 157,A -97.2481,B 15.4644,C -0.0371,E1 15.4454,E2 186.5151} C_DIS
LIN {X -13.2799,Y -129.3465,Z 157,A -95.576,B 15.4644,C -0.0393,E1 15.4501,E2 184.8329} C_DIS
LIN {X -9.3764,Y -129.6865,Z 157,A -93.9044,B 15.4644,C -0.0375,E1 15.4547,E2 183.1671} C_DIS
LIN {X -5.7243,Y -129.9006,Z 157,A -92.1912,B 15.4644,C -0.0407,E1 15.4595,E2 181.4413} C_DIS
LIN {X -1.8283,Y -130.0126,Z 157,A -90.57,B 15.4644,C -0.0378,E1 15.464,E2 179.8308} C_DIS
LIN {X 0.9057,Y -130.0191,Z 157,A -89.5983,B 15.4645,C -0.0306,E1 15.4666,E2 178.886} C_DIS
Enddeposition()
LIN {X 0.9057,Y -130.0191,Z 157,A -89.5983,B 15.4645,C -0.0306,E1 15.4666,E2 178.886} C_DIS
Startdeposition()
$VEL.CP = VEL_PRINT
LIN {X -0.0055,Y -129.0955,Z 157,A -90.6124,B 15.4647,C -0.0211,E1 15.4639,E2 179.9357} C_DIS
LIN {X -4.1786,Y -129.0273,Z 157,A -92.2828,B 15.4647,C -0.0266,E1 15.4593,E2 181.5857} C_DIS
LIN {X -7.914,Y -128.8507,Z 157,A -93.9642,B 15.4647,C -0.026,E1 15.4546,E2 183.2702} C_DIS
LIN {X -11.6556,Y -128.568,Z 157,A -95.7601,B 15.4647,C -0.0221,E1 15.4495,E2 185.082} C_DIS
LIN {X -15.8036,Y -128.1234,Z 157,A -97.4949,B 15.4647,C -0.026,E1 15.4448,E2 186.8038} C_DIS
LIN {X -20.0199,Y -127.5318,Z 157,A -99.4425,B 15.4647,C -0.0248,E1 15.4394,E2 188.7587} C_DIS
LIN {X -24.2283,Y -126.7993,Z 157,A -101.3365,B 15.4647,C -0.0256,E1 15.4341,E2 190.6529} C_DIS
LIN {X -27.749,Y -126.0767,Z 157,A -102.8644,B 15.4647,C -0.0284,E1 15.43,E2 192.1735} C_DIS
LIN {X -30.8244,Y -125.3606,Z 157,A -104.2418,B 15.4647,C -0.0299,E1 15.4263,E2 193.5483} C_DIS
LIN {X -33.799,Y -124.5913,Z 157,A -105.6128,B 15.4647,C -0.0305,E1 15.4226,E2 194.9203} C_DIS
LIN {X -36.9192,Y -123.7032,Z 157,A -107.231,B 15.4647,C -0.0261,E1 15.4182,E2 196.5594} C_DIS
LIN {X -40.4954,Y -122.5775,Z 157,A -108.8698,B 15.4647,C -0.0282,E1 15.4138,E2 198.1954} C_DIS
LIN {X -44.4425,Y -121.2039,Z 157,A -110.7298,B 15.4647,C -0.0296,E1 15.4089,E2 200.0561} C_DIS
LIN {X -47.7408,Y -119.9423,Z 157,A -112.273,B 15.4647,C -0.0319,E1 15.4049,E2 201.5964} C_DIS
LIN {X -50.9154,Y -118.6286,Z 157,A -113.8314,B 15.4647,C -0.0324,E1 15.4009,E2 203.1587} C_DIS
LIN {X -54.6494,Y -116.956,Z 157,A -115.5462,B 15.4647,C -0.0375,E1 15.3966,E2 204.8616} C_DIS
LIN {X -57.5361,Y -115.563,Z 157,A -117.0652,B 15.4647,C -0.0363,E1 15.3927,E2 206.3916} C_DIS
LIN {X -60.8577,Y -113.8505,Z 157,A -118.628,B 15.4647,C -0.0412,E1 15.3889,E2 207.9432} C_DIS
LIN {X -63.6314,Y -112.3241,Z 157,A -120.0431,B 15.4647,C -0.0428,E1 15.3854,E2 209.3592} C_DIS
LIN {X -66.4165,Y -110.7,Z 157,A -121.6056,B 15.4647,C -0.041,E1 15.3817,E2 210.9365} C_DIS
LIN {X -69.9296,Y -108.515,Z 157,A -123.3309,B 15.4647,C -0.0469,E1 15.3776,E2 212.6486} C_DIS
LIN {X -73.0395,Y -106.4459,Z 157,A -125.0978,B 15.4647,C -0.0464,E1 15.3735,E2 214.4275} C_DIS
LIN {X -76.4413,Y -104.03,Z 157,A -126.9606,B 15.4647,C -0.0491,E1 15.3693,E2 216.291} C_DIS
LIN {X -80.0461,Y -101.2832,Z 157,A -128.9458,B 15.4647,C -0.0533,E1 15.3649,E2 218.2724} C_DIS
LIN {X -83.1208,Y -98.7749,Z 157,A -130.7499,B 15.4647,C -0.0553,E1 15.361,E2 220.0807} C_DIS
LIN {X -86.0522,Y -96.2316,Z 157,A -132.4865,B 15.4647,C -0.0581,E1 15.3574,E2 221.8181} C_DIS
LIN {X -89.2189,Y -93.3032,Z 157,A -134.3976,B 15.4646,C -0.062,E1 15.3535,E2 223.7279} C_DIS
LIN {X -92.3867,Y -90.1682,Z 157,A -136.3684,B 15.4646,C -0.0662,E1 15.3496,E2 225.6967} C_DIS
LIN {X -94.589,Y -87.8547,Z 157,A -137.8282,B 15.4646,C -0.068,E1 15.3468,E2 227.1606} C_DIS
LIN {X -97.4241,Y -84.7001,Z 157,A -139.7298,B 15.4646,C -0.0715,E1 15.3433,E2 229.0632} C_DIS
LIN {X -99.9196,Y -81.7409,Z 157,A -141.3558,B 15.4646,C -0.078,E1 15.3404,E2 230.6775} C_DIS
LIN {X -102.2586,Y -78.7961,Z 157,A -143.2049,B 15.4646,C -0.0767,E1 15.3372,E2 232.5462} C_DIS
LIN {X -104.8763,Y -75.2763,Z 157,A -145.123,B 15.4645,C -0.0821,E1 15.334,E2 234.4595} C_DIS
LIN {X -107.3481,Y -71.707,Z 157,A -147.0482,B 15.4645,C -0.0868,E1 15.331,E2 236.383} C_DIS
LIN {X -109.6053,Y -68.207,Z 157,A -148.9136,B 15.4645,C -0.0909,E1 15.3282,E2 238.2489} C_DIS
LIN {X -111.7559,Y -64.6229,Z 157,A -150.79,B 15.4645,C -0.095,E1 15.3256,E2 240.1261} C_DIS
LIN {X -113.5806,Y -61.36,Z 157,A -152.4306,B 15.4644,C -0.0998,E1 15.3234,E2 241.7632} C_DIS
LIN {X -115.0476,Y -58.558,Z 157,A -153.8616,B 15.4644,C -0.1028,E1 15.3215,E2 243.196} C_DIS
LIN {X -116.7057,Y -55.182,Z 157,A -155.4594,B 15.4644,C -0.1092,E1 15.3196,E2 244.7841} C_DIS
LIN {X -118.021,Y -52.309,Z 157,A -156.8731,B 15.4644,C -0.1127,E1 15.318,E2 246.1978} C_DIS
LIN {X -119.2662,Y -49.4036,Z 157,A -158.2879,B 15.4643,C -0.1162,E1 15.3164,E2 247.6125} C_DIS
LIN {X -120.4401,Y -46.4684,Z 157,A -159.7031,B 15.4643,C -0.1197,E1 15.315,E2 249.0277} C_DIS
LIN {X -121.6267,Y -43.2697,Z 157,A -161.4057,B 15.4643,C -0.1188,E1 15.3134,E2 250.7503} C_DIS
LIN {X -122.9757,Y -39.2685,Z 157,A -163.1726,B 15.4642,C -0.127,E1 15.3118,E2 252.5031} C_DIS
LIN {X -123.9861,Y -35.9528,Z 157,A -164.6748,B 15.4642,C -0.1324,E1 15.3106,E2 253.9995} C_DIS
LIN {X -124.8304,Y -32.9023,Z 157,A -166.0923,B 15.4642,C -0.1361,E1 15.3096,E2 255.4169} C_DIS
LIN {X -125.5997,Y -29.8322,Z 157,A -167.5092,B 15.4641,C -0.1399,E1 15.3087,E2 256.8337} C_DIS
LIN {X -126.4156,Y -26.1601,Z 157,A -169.3044,B 15.4641,C -0.1413,E1 15.3076,E2 258.6414} C_DIS
LIN {X -127.1807,Y -22.1475,Z 157,A -171.0233,B 15.4641,C -0.1492,E1 15.3067,E2 260.3475} C_DIS
LIN {X -127.6976,Y -18.9449,Z 157,A -172.4449,B 15.464,C -0.154,E1 15.3061,E2 261.7653} C_DIS
LIN {X -128.1243,Y -15.7966,Z 157,A -174.0464,B 15.464,C -0.153,E1 15.3056,E2 263.3869} C_DIS
LIN {X -128.5717,Y -11.6167,Z 157,A -175.9542,B 15.464,C -0.1574,E1 15.305,E2 265.2973} C_DIS
LIN {X -128.8508,Y -7.9122,Z 157,A -177.5262,B 15.4639,C -0.1645,E1 15.3047,E2 266.8585} C_DIS
LIN {X -129.0269,Y -4.1931,Z 157,A -179.2525,B 15.4639,C -0.1674,E1 15.3046,E2 268.5912} C_DIS
LIN {X -129.0967,Y -0.0367,Z 157,A 178.8168,B 15.4638,C -0.1706,E1 15.3046,E2 270.5294} C_DIS
LIN {X -129.0271,Y 4.1855,Z 157,A 177.133,B 15.4637,C -0.1815,E1 15.3046,E2 272.1891} C_DIS
LIN {X -128.8509,Y 7.9103,Z 157,A 175.4366,B 15.4637,C -0.1854,E1 15.3049,E2 273.8881} C_DIS
LIN {X -128.5669,Y 11.6669,Z 157,A 173.6208,B 15.4637,C -0.1865,E1 15.3053,E2 275.7181} C_DIS
LIN {X -128.1908,Y 15.2386,Z 157,A 172.0591,B 15.4635,C -0.1922,E1 15.3058,E2 277.274} C_DIS
LIN {X -127.7792,Y 18.3732,Z 157,A 170.6587,B 15.4635,C -0.1965,E1 15.3063,E2 278.6723} C_DIS
LIN {X -127.1959,Y 22.0627,Z 157,A 168.8858,B 15.4635,C -0.1984,E1 15.3071,E2 280.4561} C_DIS
LIN {X -126.4132,Y 26.1721,Z 157,A 167.1775,B 15.4633,C -0.208,E1 15.308,E2 282.1451} C_DIS
LIN {X -125.7322,Y 29.2705,Z 157,A 165.755,B 15.4633,C -0.2117,E1 15.3089,E2 283.5674} C_DIS
LIN {X -125.0839,Y 31.9235,Z 157,A 164.4752,B 15.4633,C -0.2135,E1 15.3098,E2 284.8532} C_DIS
LIN {X -124.264,Y 34.9793,Z 157,A 163.0597,B 15.4633,C -0.2173,E1 15.3108,E2 286.2681} C_DIS
LIN {X -123.0682,Y 38.979,Z 157,A 161.2355,B 15.4631,C -0.2235,E1 15.3123,E2 288.0866} C_DIS
LIN {X -121.884,Y 42.5369,Z 157,A 159.5116,B 15.4631,C -0.2267,E1 15.3139,E2 289.815} C_DIS
LIN {X -120.6444,Y 45.9396,Z 157,A 157.9292,B 15.4631,C -0.232,E1 15.3154,E2 291.3925} C_DIS
LIN {X -119.6462,Y 48.4753,Z 157,A 156.6589,B 15.463,C -0.2338,E1 15.3167,E2 292.668} C_DIS
LIN {X -118.0184,Y 52.3149,Z 157,A 154.9333,B 15.4629,C -0.2425,E1 15.3186,E2 294.3769} C_DIS
LIN {X -116.619,Y 55.3634,Z 157,A 153.4571,B 15.4628,C -0.247,E1 15.3204,E2 295.8497} C_DIS
LIN {X -115.4567,Y 57.7517,Z 157,A 152.0449,B 15.4628,C -0.2438,E1 15.3221,E2 297.2869} C_DIS
LIN {X -113.5494,Y 61.418,Z 157,A 150.1835,B 15.4628,C -0.248,E1 15.3246,E2 299.1488} C_DIS
LIN {X -111.5468,Y 64.9841,Z 157,A 148.4577,B 15.4627,C -0.2554,E1 15.3269,E2 300.8622} C_DIS
LIN {X -109.6011,Y 68.2137,Z 157,A 146.7048,B 15.4627,C -0.2576,E1 15.3295,E2 302.6218} C_DIS
LIN {X -107.658,Y 71.2415,Z 157,A 145.1622,B 15.4625,C -0.2632,E1 15.3318,E2 304.1562} C_DIS
LIN {X -105.8794,Y 73.8586,Z 157,A 143.6315,B 15.4625,C -0.2633,E1 15.3343,E2 305.6994} C_DIS
LIN {X -103.686,Y 76.9076,Z 157,A 141.9163,B 15.4625,C -0.2661,E1 15.3371,E2 307.4179} C_DIS
LIN {X -100.7894,Y 80.6667,Z 157,A 139.8328,B 15.4624,C -0.2719,E1 15.3407,E2 309.4961} C_DIS
LIN {X -98.2587,Y 83.7303,Z 157,A 138.0703,B 15.4624,C -0.2762,E1 15.3439,E2 311.2562} C_DIS
LIN {X -95.6484,Y 86.7001,Z 157,A 136.3087,B 15.4622,C -0.2801,E1 15.3471,E2 313.0164} C_DIS
LIN {X -92.948,Y 89.5893,Z 157,A 134.5223,B 15.4622,C -0.2832,E1 15.3506,E2 314.8041} C_DIS
LIN {X -90.1605,Y 92.3942,Z 157,A 132.7979,B 15.4621,C -0.2879,E1 15.354,E2 316.523} C_DIS
LIN {X -87.2751,Y 95.124,Z 157,A 131.0369,B 15.4621,C -0.2917,E1 15.3576,E2 318.2816} C_DIS
LIN {X -84.3209,Y 97.7523,Z 157,A 129.2602,B 15.462,C -0.2947,E1 15.3613,E2 320.0587} C_DIS
LIN {X -81.2865,Y 100.2901,Z 157,A 127.4537,B 15.462,C -0.2968,E1 15.3652,E2 321.8689} C_DIS
LIN {X -78.1648,Y 102.7418,Z 157,A 125.6517,B 15.4619,C -0.2991,E1 15.3692,E2 323.6734} C_DIS
LIN {X -74.8042,Y 105.2139,Z 157,A 123.9081,B 15.4618,C -0.3056,E1 15.3731,E2 325.4027} C_DIS
LIN {X -71.7252,Y 107.3359,Z 157,A 122.2458,B 15.4618,C -0.3085,E1 15.3769,E2 327.0635} C_DIS
LIN {X -69.0729,Y 109.0618,Z 157,A 120.8349,B 15.4617,C -0.3107,E1 15.3803,E2 328.4737} C_DIS
LIN {X -65.9637,Y 110.9699,Z 157,A 119.0884,B 15.4617,C -0.3097,E1 15.3845,E2 330.2328} C_DIS
LIN {X -62.724,Y 112.8329,Z 157,A 117.5404,B 15.4616,C -0.3155,E1 15.3882,E2 331.7667} C_DIS
LIN {X -59.9497,Y 114.3286,Z 157,A 116.1298,B 15.4616,C -0.3173,E1 15.3917,E2 333.1771} C_DIS
LIN {X -56.6199,Y 116.015,Z 157,A 114.3509,B 15.4616,C -0.3162,E1 15.3961,E2 334.9682} C_DIS
LIN {X -52.8449,Y 117.7813,Z 157,A 112.5043,B 15.4616,C -0.3188,E1 15.4008,E2 336.8127} C_DIS
LIN {X -49.4141,Y 119.2619,Z 157,A 110.9373,B 15.4614,C -0.3235,E1 15.4048,E2 338.3677} C_DIS
LIN {X -46.4599,Y 120.4434,Z 157,A 109.4432,B 15.4614,C -0.3228,E1 15.4087,E2 339.8698} C_DIS
LIN {X -42.5175,Y 121.8908,Z 157,A 107.6526,B 15.4614,C -0.3271,E1 15.4134,E2 341.6505} C_DIS
LIN {X -39.5196,Y 122.8955,Z 157,A 106.1345,B 15.4614,C -0.3252,E1 15.4175,E2 343.1804} C_DIS
LIN {X -35.9507,Y 123.9867,Z 157,A 104.5841,B 15.4613,C -0.3298,E1 15.4216,E2 344.7175} C_DIS
LIN {X -32.9024,Y 124.8304,Z 157,A 103.1753,B 15.4613,C -0.3309,E1 15.4254,E2 346.1258} C_DIS
LIN {X -29.819,Y 125.6029,Z 157,A 101.7643,B 15.4613,C -0.3321,E1 15.4292,E2 347.5357} C_DIS
LIN {X -26.1227,Y 126.4232,Z 157,A 99.9774,B 15.4613,C -0.3302,E1 15.4341,E2 349.3335} C_DIS
LIN {X -22.0563,Y 127.197,Z 157,A 98.2458,B 15.4612,C -0.3345,E1 15.4388,E2 351.0519} C_DIS
LIN {X -18.9482,Y 127.6971,Z 157,A 96.8233,B 15.4612,C -0.3345,E1 15.4428,E2 352.4764} C_DIS
LIN {X -15.8275,Y 128.1206,Z 157,A 95.2974,B 15.4612,C -0.3314,E1 15.447,E2 354.0159} C_DIS
LIN {X -11.6486,Y 128.5687,Z 157,A 93.4083,B 15.4612,C -0.3314,E1 15.4523,E2 355.9065} C_DIS
LIN {X -7.919,Y 128.8504,Z 157,A 91.9016,B 15.4612,C -0.3365,E1 15.4564,E2 357.3949} C_DIS
LIN {X -4.1693,Y 129.0275,Z 157,A 90.1167,B 15.4612,C -0.3333,E1 15.4614,E2 359.1924} C_DIS
LIN {X 0.0022,Y 129.0956,Z 157,A 88.2218,B 15.4612,C -0.3322,E1 15.4667,E2 361.0913} C_DIS
LIN {X 4.1727,Y 129.0274,Z 157,A 86.5638,B 15.4612,C -0.3381,E1 15.4713,E2 362.7265} C_DIS
LIN {X 6.7474,Y 128.9173,Z 157,A 85.2809,B 15.4612,C -0.3338,E1 15.4749,E2 364.0248} C_DIS
LIN {X 11.0777,Y 128.6175,Z 157,A 83.4008,B 15.4612,C -0.335,E1 15.4801,E2 365.8989} C_DIS
LIN {X 15.2814,Y 128.1857,Z 157,A 81.5155,B 15.4612,C -0.3343,E1 15.4854,E2 367.7846} C_DIS
LIN {X 18.3885,Y 127.7771,Z 157,A 80.1482,B 15.4612,C -0.3345,E1 15.4892,E2 369.1488} C_DIS
LIN {X 22.0969,Y 127.1898,Z 157,A 78.381,B 15.4612,C -0.3308,E1 15.4941,E2 370.9271} C_DIS
LIN {X 26.1927,Y 126.409,Z 157,A 76.6926,B 15.4612,C -0.3349,E1 15.4986,E2 372.5966} C_DIS
LIN {X 29.2781,Y 125.7305,Z 157,A 75.3058,B 15.4612,C -0.3345,E1 15.5024,E2 373.9814} C_DIS
LIN {X 31.9255,Y 125.0834,Z 157,A 74.031,B 15.4612,C -0.3318,E1 15.5059,E2 375.2633} C_DIS
LIN {X 34.9778,Y 124.2644,Z 157,A 72.6328,B 15.4612,C -0.3309,E1 15.5096,E2 376.6609} C_DIS
LIN {X 38.8599,Y 123.1062,Z 157,A 70.8479,B 15.4612,C -0.3299,E1 15.5144,E2 378.4442} C_DIS
LIN {X 42.5404,Y 121.8828,Z 157,A 69.1256,B 15.4613,C -0.3284,E1 15.519,E2 380.1665} C_DIS
LIN {X 45.9223,Y 120.6509,Z 157,A 67.5762,B 15.4613,C -0.3284,E1 15.523,E2 381.7104} C_DIS
LIN {X 49.3938,Y 119.2704,Z 157,A 66.0879,B 15.4613,C -0.332,E1 15.5268,E2 383.1793} C_DIS
LIN {X 52.8522,Y 117.7781,Z 157,A 64.2028,B 15.4614,C -0.3233,E1 15.5317,E2 385.089} C_DIS
LIN {X 56.113,Y 116.2609,Z 157,A 62.6657,B 15.4614,C -0.3233,E1 15.5355,E2 386.6194} C_DIS
LIN {X 59.4541,Y 114.5888,Z 157,A 61.044,B 15.4614,C -0.3223,E1 15.5396,E2 388.2373} C_DIS
LIN {X 62.2464,Y 113.0973,Z 157,A 59.627,B 15.4614,C -0.32,E1 15.5431,E2 389.6559} C_DIS
LIN {X 64.9991,Y 111.5382,Z 157,A 58.1569,B 15.4616,C -0.3159,E1 15.5466,E2 391.1338} C_DIS
LIN {X 68.2377,Y 109.5862,Z 157,A 56.4864,B 15.4616,C -0.3137,E1 15.5506,E2 392.8039} C_DIS
LIN {X 71.2505,Y 107.6521,Z 157,A 54.8509,B 15.4616,C -0.3097,E1 15.5545,E2 394.4451} C_DIS
LIN {X 74.8057,Y 105.2128,Z 157,A 52.973,B 15.4617,C -0.3077,E1 15.5587,E2 396.3195} C_DIS
LIN {X 77.7098,Y 103.0859,Z 157,A 51.4266,B 15.4617,C -0.3066,E1 15.5622,E2 397.8607} C_DIS
LIN {X 80.675,Y 100.7828,Z 157,A 49.7142,B 15.4618,C -0.3021,E1 15.566,E2 399.579} C_DIS
LIN {X 83.7209,Y 98.2667,Z 157,A 47.9889,B 15.4618,C -0.2998,E1 15.5697,E2 401.3018} C_DIS
LIN {X 86.6892,Y 95.6582,Z 157,A 46.2513,B 15.4619,C -0.2969,E1 15.5733,E2 403.0385} C_DIS
LIN {X 89.5887,Y 92.9487,Z 157,A 44.4639,B 15.462,C -0.2925,E1 15.5769,E2 404.8298} C_DIS
LIN {X 92.6098,Y 89.9386,Z 157,A 42.6125,B 15.462,C -0.29,E1 15.5805,E2 406.6775} C_DIS
LIN {X 95.4644,Y 86.9028,Z 157,A 40.7647,B 15.4621,C -0.286,E1 15.584,E2 408.5262} C_DIS
LIN {X 98.2652,Y 83.7226,Z 157,A 38.96,B 15.4621,C -0.2844,E1 15.5873,E2 410.3233} C_DIS
LIN {X 100.7919,Y 80.6636,Z 157,A 37.1049,B 15.4623,C -0.2773,E1 15.5906,E2 412.1904} C_DIS
LIN {X 103.3746,Y 77.3258,Z 157,A 35.2927,B 15.4623,C -0.2749,E1 15.5937,E2 413.997} C_DIS
LIN {X 105.4268,Y 74.503,Z 157,A 33.7858,B 15.4623,C -0.2726,E1 15.5961,E2 415.5002} C_DIS
LIN {X 107.7125,Y 71.1587,Z 157,A 31.9418,B 15.4625,C -0.2666,E1 15.599,E2 417.3508} C_DIS
LIN {X 110.2119,Y 67.2231,Z 157,A 29.9355,B 15.4625,C -0.2635,E1 15.6019,E2 419.3516} C_DIS
LIN {X 112.0415,Y 64.1268,Z 157,A 28.4503,B 15.4625,C -0.2632,E1 15.604,E2 420.8253} C_DIS
LIN {X 113.579,Y 61.363,Z 157,A 26.98,B 15.4626,C -0.2573,E1 15.606,E2 422.3045} C_DIS
LIN {X 115.046,Y 58.5612,Z 157,A 25.5791,B 15.4626,C -0.2537,E1 15.6078,E2 423.7063} C_DIS
LIN {X 116.7687,Y 55.0501,Z 157,A 23.9414,B 15.4627,C -0.2523,E1 15.6098,E2 425.3343} C_DIS
LIN {X 118.0226,Y 52.3056,Z 157,A 22.6138,B 15.4627,C -0.2491,E1 15.6113,E2 426.6618} C_DIS
LIN {X 119.2674,Y 49.4008,Z 157,A 21.2247,B 15.4628,C -0.2457,E1 15.6128,E2 428.0507} C_DIS
LIN {X 120.4435,Y 46.4597,Z 157,A 19.7559,B 15.4628,C -0.2397,E1 15.6143,E2 429.5281} C_DIS
LIN {X 121.8823,Y 42.5419,Z 157,A 17.9973,B 15.4629,C -0.2376,E1 15.616,E2 431.2778} C_DIS
LIN {X 122.8906,Y 39.535,Z 157,A 16.4928,B 15.463,C -0.2304,E1 15.6173,E2 432.795} C_DIS
LIN {X 123.9865,Y 35.9514,Z 157,A 14.8803,B 15.463,C -0.2273,E1 15.6186,E2 434.4033} C_DIS
LIN {X 125.0825,Y 31.9289,Z 157,A 13.0135,B 15.4632,C -0.2214,E1 15.6199,E2 436.2741} C_DIS
LIN {X 125.9717,Y 28.2222,Z 157,A 11.3267,B 15.4632,C -0.2166,E1 15.621,E2 437.9622} C_DIS
LIN {X 126.8104,Y 24.1706,Z 157,A 9.5691,B 15.4632,C -0.2139,E1 15.6219,E2 439.7127} C_DIS
LIN {X 127.3607,Y 21.0798,Z 157,A 8.1859,B 15.4633,C -0.2101,E1 15.6226,E2 441.0964} C_DIS
LIN {X 127.9116,Y 17.4408,Z 157,A 6.598,B 15.4633,C -0.2068,E1 15.6232,E2 442.681} C_DIS
LIN {X 128.3688,Y 13.6598,Z 157,A 4.9186,B 15.4634,C -0.2021,E1 15.6237,E2 444.3611} C_DIS
LIN {X 128.7434,Y 9.5015,Z 157,A 3.1456,B 15.4634,C -0.1992,E1 15.6241,E2 446.127} C_DIS
LIN {X 128.9671,Y 5.7581,Z 157,A 1.4566,B 15.4635,C -0.1934,E1 15.6244,E2 447.821} C_DIS
LIN {X 129.0754,Y 2.1631,Z 157,A -0.1375,B 15.4635,C -0.1886,E1 15.6244,E2 449.4167} C_DIS
LIN {X 129.0852,Y -1.5767,Z 157,A -1.9024,B 15.4637,C -0.18,E1 15.6244,E2 451.196} C_DIS
LIN {X 128.9918,Y -5.1245,Z 157,A -3.3495,B 15.4637,C -0.1796,E1 15.6244,E2 452.6301} C_DIS
LIN {X 128.7674,Y -9.1723,Z 157,A -5.0694,B 15.4637,C -0.1769,E1 15.624,E2 454.3431} C_DIS
LIN {X 128.466,Y -12.7182,Z 157,A -6.6386,B 15.4637,C -0.1724,E1 15.6236,E2 455.9131} C_DIS
LIN {X 128.049,Y -16.3923,Z 157,A -8.3693,B 15.4639,C -0.1644,E1 15.6231,E2 457.6564} C_DIS
LIN {X 127.5398,Y -19.9686,Z 157,A -9.9368,B 15.4639,C -0.1608,E1 15.6224,E2 459.2219} C_DIS
LIN {X 126.8055,Y -24.196,Z 157,A -11.8168,B 15.4639,C -0.1559,E1 15.6215,E2 461.1016} C_DIS
LIN {X 126.0795,Y -27.7361,Z 157,A -13.3306,B 15.4639,C -0.1542,E1 15.6206,E2 462.607} C_DIS
LIN {X 125.4286,Y -30.542,Z 157,A -14.5788,B 15.4639,C -0.1514,E1 15.6198,E2 463.8533} C_DIS
LIN {X 124.5731,Y -33.8674,Z 157,A -16.085,B 15.464,C -0.1475,E1 15.6187,E2 465.3596} C_DIS
LIN {X 123.7,Y -36.93,Z 157,A -17.6573,B 15.4641,C -0.1379,E1 15.6175,E2 466.9524} C_DIS
LIN {X 122.5779,Y -40.4944,Z 157,A -19.2682,B 15.4641,C -0.1347,E1 15.6161,E2 468.5599} C_DIS
LIN {X 121.1767,Y -44.5178,Z 157,A -21.0276,B 15.4641,C -0.1336,E1 15.6145,E2 470.3066} C_DIS
LIN {X 120.0612,Y -47.4431,Z 157,A -22.3924,B 15.4641,C -0.1305,E1 15.6131,E2 471.6702} C_DIS
LIN {X 118.8702,Y -50.3518,Z 157,A -23.7645,B 15.4641,C -0.1273,E1 15.6116,E2 473.0415} C_DIS
LIN {X 117.533,Y -53.4002,Z 157,A -25.2508,B 15.4642,C -0.1228,E1 15.6099,E2 474.5309} C_DIS
LIN {X 116.2724,Y -56.089,Z 157,A -26.5572,B 15.4642,C -0.1195,E1 15.6084,E2 475.8376} C_DIS
LIN {X 114.5888,Y -59.4541,Z 157,A -28.1833,B 15.4642,C -0.1164,E1 15.6063,E2 477.4609} C_DIS
LIN {X 113.0975,Y -62.2462,Z 157,A -29.5941,B 15.4643,C -0.1124,E1 15.6044,E2 478.8743} C_DIS
LIN {X 111.5276,Y -65.0174,Z 157,A -31.0054,B 15.4643,C -0.1086,E1 15.6025,E2 480.2872} C_DIS
LIN {X 109.598,Y -68.2186,Z 157,A -32.7156,B 15.4643,C -0.1025,E1 15.6,E2 482.0057} C_DIS
LIN {X 107.6556,Y -71.2451,Z 157,A -34.3481,B 15.4644,C -0.0971,E1 15.5975,E2 483.6445} C_DIS
LIN {X 105.1949,Y -74.8307,Z 157,A -36.234,B 15.4644,C -0.0936,E1 15.5944,E2 485.5278} C_DIS
LIN {X 102.7337,Y -78.1753,Z 157,A -38.0884,B 15.4644,C -0.0886,E1 15.5913,E2 487.3859} C_DIS
LIN {X 100.1104,Y -81.5075,Z 157,A -39.936,B 15.4644,C -0.0851,E1 15.5881,E2 489.2318} C_DIS
LIN {X 97.3981,Y -84.7299,Z 157,A -41.748,B 15.4644,C -0.0826,E1 15.5848,E2 491.0396} C_DIS
LIN {X 94.765,Y -87.6657,Z 157,A -43.4931,B 15.4645,C -0.0786,E1 15.5816,E2 492.7862} C_DIS
LIN {X 92.0419,Y -90.5198,Z 157,A -45.208,B 15.4645,C -0.0759,E1 15.5782,E2 494.4991} C_DIS
LIN {X 89.2024,Y -93.319,Z 157,A -46.9721,B 15.4645,C -0.0721,E1 15.5747,E2 496.2647} C_DIS
LIN {X 86.3083,Y -96.0023,Z 157,A -48.7717,B 15.4645,C -0.0667,E1 15.571,E2 498.072} C_DIS
LIN {X 83.1132,Y -98.7812,Z 157,A -50.6222,B 15.4645,C -0.0638,E1 15.567,E2 499.9213} C_DIS
LIN {X 80.0327,Y -101.2937,Z 157,A -52.4357,B 15.4646,C -0.0586,E1 15.5631,E2 501.7428} C_DIS
LIN {X 76.431,Y -104.0375,Z 157,A -54.3478,B 15.4646,C -0.0579,E1 15.5588,E2 503.6457} C_DIS
LIN {X 73.5042,Y -106.126,Z 157,A -55.9802,B 15.4646,C -0.0537,E1 15.5551,E2 505.2842} C_DIS
LIN {X 70.4022,Y -108.2084,Z 157,A -57.5057,B 15.4646,C -0.0551,E1 15.5516,E2 506.7959} C_DIS
LIN {X 67.2255,Y -110.2104,Z 157,A -59.2599,B 15.4646,C -0.0494,E1 15.5474,E2 508.5623} C_DIS
LIN {X 64.1301,Y -112.0396,Z 157,A -60.8058,B 15.4646,C -0.0484,E1 15.5436,E2 510.104} C_DIS
LIN {X 61.2224,Y -113.6545,Z 157,A -62.2758,B 15.4646,C -0.0462,E1 15.54,E2 511.5747} C_DIS
LIN {X 58.4961,Y -115.0791,Z 157,A -63.6563,B 15.4646,C -0.0437,E1 15.5366,E2 512.9583} C_DIS
LIN {X 55.2057,Y -116.6943,Z 157,A -65.2042,B 15.4646,C -0.0439,E1 15.5327,E2 514.4986} C_DIS
LIN {X 52.3207,Y -118.0158,Z 157,A -66.605,B 15.4646,C -0.0421,E1 15.5292,E2 515.8999} C_DIS
LIN {X 49.3946,Y -119.27,Z 157,A -68.0089,B 15.4646,C -0.0406,E1 15.5256,E2 517.304} C_DIS
LIN {X 46.4559,Y -120.4449,Z 157,A -69.4858,B 15.4646,C -0.0365,E1 15.5217,E2 518.7906} C_DIS
LIN {X 42.538,Y -121.8837,Z 157,A -71.2659,B 15.4646,C -0.0366,E1 15.517,E2 520.564} C_DIS
LIN {X 39.4914,Y -122.9045,Z 157,A -72.7755,B 15.4646,C -0.0324,E1 15.513,E2 522.0845} C_DIS
LIN {X 35.9367,Y -123.9908,Z 157,A -74.4052,B 15.4646,C -0.0314,E1 15.5086,E2 523.7133} C_DIS
LIN {X 31.9194,Y -125.0849,Z 157,A -76.1549,B 15.4646,C -0.0328,E1 15.5039,E2 525.453} C_DIS
LIN {X 28.2243,Y -125.9712,Z 157,A -77.9596,B 15.4646,C -0.0276,E1 15.499,E2 527.2728} C_DIS
LIN {X 24.1922,Y -126.8062,Z 157,A -79.7316,B 15.4646,C -0.028,E1 15.4941,E2 529.0396} C_DIS
LIN {X 20.5635,Y -127.4469,Z 157,A -81.2812,B 15.4646,C -0.0296,E1 15.4899,E2 530.5803} C_DIS
LIN {X 17.3763,Y -127.92,Z 157,A -82.7378,B 15.4646,C -0.028,E1 15.4859,E2 532.041} C_DIS
LIN {X 13.651,Y -128.3697,Z 157,A -84.4255,B 15.4646,C -0.0264,E1 15.4812,E2 533.7323} C_DIS
LIN {X 9.4951,Y -128.7438,Z 157,A -86.2353,B 15.4646,C -0.027,E1 15.4762,E2 535.5382} C_DIS
LIN {X 6.3351,Y -128.9381,Z 157,A -87.6703,B 15.4646,C -0.0256,E1 15.4721,E2 536.9775} C_DIS
LIN {X 2.2309,Y -129.0743,Z 157,A -89.5448,B 15.4646,C -0.0236,E1 15.4669,E2 538.859} C_DIS
LIN {X 2.2309,Y -129.0743,Z 157,A -89.5448,B 15.4646,C -0.0236,E1 15.4669,E2 538.859} C_DIS
Enddeposition()
LIN {X 0.9594,Y -136.8014,Z 158,A -92.6497,B 24.9706,C -1.2534,E1 25.0012,E2 539.3202} C_DIS
Startdeposition()
$VEL.CP = VEL_PRINT
LIN {X 7.5032,Y -136.6001,Z 158,A -89.5657,B 24.9697,C -1.2729,E1 25.01,E2 536.1907} C_DIS
LIN {X 13.5162,Y -136.1359,Z 158,A -86.941,B 24.9693,C -1.2796,E1 25.0173,E2 533.5514} C_DIS
LIN {X 17.1604,Y -135.7253,Z 158,A -85.4827,B 24.9695,C -1.2763,E1 25.0213,E2 532.1021} C_DIS
LIN {X 20.4893,Y -135.2621,Z 158,A -84.0161,B 24.9693,C -1.2806,E1 25.0254,E2 530.6267} C_DIS
LIN {X 23.9064,Y -134.6995,Z 158,A -82.5449,B 24.9692,C -1.2829,E1 25.0294,E2 529.1517} C_DIS
LIN {X 27.7881,Y -133.9534,Z 158,A -80.8384,B 24.969,C -1.2872,E1 25.0341,E2 527.4371} C_DIS
LIN {X 31.8792,Y -133.0382,Z 158,A -79.1393,B 24.969,C -1.2858,E1 25.0387,E2 525.7437} C_DIS
LIN {X 36.2789,Y -131.9075,Z 158,A -77.3888,B 24.9693,C -1.2793,E1 25.0434,E2 524.0112} C_DIS
LIN {X 39.7404,Y -130.9052,Z 158,A -75.7177,B 24.9688,C -1.2901,E1 25.048,E2 522.3175} C_DIS
LIN {X 43.148,Y -129.8215,Z 158,A -74.2485,B 24.9688,C -1.2904,E1 25.0518,E2 520.8503} C_DIS
LIN {X 47.0197,Y -128.4716,Z 158,A -72.5655,B 24.9688,C -1.2908,E1 25.0563,E2 519.17} C_DIS
LIN {X 50.4677,Y -127.157,Z 158,A -70.936,B 24.9685,C -1.2977,E1 25.0605,E2 517.5277} C_DIS
LIN {X 54.0158,Y -125.689,Z 158,A -69.4372,B 24.9686,C -1.294,E1 25.0644,E2 516.0412} C_DIS
LIN {X 56.4495,Y -124.6163,Z 158,A -67.7261,B 24.9669,C -1.3295,E1 25.0689,E2 514.2505} C_DIS
LIN {X 60.9449,Y -122.4797,Z 158,A -66.2024,B 24.9683,C -1.3012,E1 25.0726,E2 512.7978} C_DIS
LIN {X 65.0176,Y -120.3689,Z 158,A -64.302,B 24.9682,C -1.3034,E1 25.0772,E2 510.8976} C_DIS
LIN {X 69.2492,Y -117.9849,Z 158,A -62.2421,B 24.9679,C -1.3086,E1 25.0822,E2 508.8315} C_DIS
LIN {X 73.0926,Y -115.6432,Z 158,A -60.4333,B 24.9679,C -1.3079,E1 25.0865,E2 507.0299} C_DIS
LIN {X 76.4394,Y -113.4592,Z 158,A -58.8331,B 24.9679,C -1.3072,E1 25.0902,E2 505.4369} C_DIS
LIN {X 81.0388,Y -110.2206,Z 158,A -56.3503,B 24.9674,C -1.3193,E1 25.0959,E2 502.934} C_DIS
LIN {X 84.3789,Y -107.6852,Z 158,A -54.5774,B 24.9672,C -1.3242,E1 25.0998,E2 501.1562} C_DIS
LIN {X 87.4484,Y -105.208,Z 158,A -52.8508,B 24.9668,C -1.3322,E1 25.1036,E2 499.4172} C_DIS
LIN {X 91.1603,Y -102.0083,Z 158,A -50.8924,B 24.9668,C -1.3317,E1 25.1077,E2 497.4678} C_DIS
LIN {X 94.3555,Y -99.0604,Z 158,A -49.0695,B 24.9666,C -1.3363,E1 25.1114,E2 495.6416} C_DIS
LIN {X 97.2215,Y -96.2492,Z 158,A -47.2539,B 24.966,C -1.3482,E1 25.115,E2 493.8056} C_DIS
LIN {X 100.7649,Y -92.5327,Z 158,A -45.3653,B 24.9664,C -1.3387,E1 25.1186,E2 491.9475} C_DIS
LIN {X 103.3933,Y -89.5872,Z 158,A -43.5954,B 24.9659,C -1.3497,E1 25.1219,E2 490.1596} C_DIS
LIN {X 106.3342,Y -86.0754,Z 158,A -41.703,B 24.9657,C -1.3535,E1 25.1252,E2 488.2672} C_DIS
LIN {X 108.9797,Y -82.7009,Z 158,A -39.9218,B 24.9655,C -1.3576,E1 25.1283,E2 486.4847} C_DIS
LIN {X 111.6343,Y -79.0806,Z 158,A -38.0614,B 24.9653,C -1.3618,E1 25.1313,E2 484.6234} C_DIS
LIN {X 114.1668,Y -75.378,Z 158,A -36.3593,B 24.9655,C -1.357,E1 25.1339,E2 482.9409} C_DIS
LIN {X 116.1307,Y -72.3155,Z 158,A -33.9654,B 24.9627,C -1.412,E1 25.1376,E2 480.4296} C_DIS
LIN {X 119.2635,Y -67.0232,Z 158,A -32.2438,B 24.9648,C -1.37,E1 25.1399,E2 478.8157} C_DIS
LIN {X 120.8867,Y -64.0467,Z 158,A -30.8466,B 24.9647,C -1.3731,E1 25.1417,E2 477.4188} C_DIS
LIN {X 122.3994,Y -61.1076,Z 158,A -29.4869,B 24.9645,C -1.3759,E1 25.1434,E2 476.0597} C_DIS
LIN {X 124.0315,Y -57.7205,Z 158,A -27.8536,B 24.9641,C -1.3841,E1 25.1454,E2 474.4156} C_DIS
LIN {X 126.5207,Y -52.0424,Z 158,A -25.1537,B 24.9634,C -1.3982,E1 25.1484,E2 471.6974} C_DIS
LIN {X 128.0959,Y -48.0293,Z 158,A -23.486,B 24.9634,C -1.396,E1 25.15,E2 470.0441} C_DIS
LIN {X 129.4472,Y -44.2621,Z 158,A -21.8356,B 24.9633,C -1.3999,E1 25.1516,E2 468.3939} C_DIS
LIN {X 130.6375,Y -40.6151,Z 158,A -20.2719,B 24.9631,C -1.4026,E1 25.1529,E2 466.8326} C_DIS
LIN {X 131.5684,Y -37.4914,Z 158,A -18.7827,B 24.9625,C -1.4142,E1 25.1541,E2 465.3246} C_DIS
LIN {X 132.579,Y -33.7376,Z 158,A -17.2918,B 24.9627,C -1.4116,E1 25.1551,E2 463.8485} C_DIS
LIN {X 133.349,Y -30.5524,Z 158,A -15.9369,B 24.9625,C -1.4151,E1 25.156,E2 462.4931} C_DIS
LIN {X 134.0367,Y -27.3785,Z 158,A -14.4745,B 24.9619,C -1.4255,E1 25.1568,E2 461.0147} C_DIS
LIN {X 134.8791,Y -22.8734,Z 158,A -12.6274,B 24.9619,C -1.4277,E1 25.1577,E2 459.1734} C_DIS
LIN {X 135.413,Y -19.4622,Z 158,A -11.196,B 24.9616,C -1.4316,E1 25.1583,E2 457.7411} C_DIS
LIN {X 135.8869,Y -15.8227,Z 158,A -9.5495,B 24.961,C -1.4431,E1 25.1589,E2 456.0773} C_DIS
LIN {X 136.341,Y -11.2547,Z 158,A -7.6959,B 24.9609,C -1.4455,E1 25.1593,E2 454.2292} C_DIS
LIN {X 136.6116,Y -7.2742,Z 158,A -5.9654,B 24.9604,C -1.4545,E1 25.1596,E2 452.4877} C_DIS
LIN {X 136.7571,Y -3.6071,Z 158,A -4.3903,B 24.96,C -1.4618,E1 25.1598,E2 450.9046} C_DIS
LIN {X 136.7999,Y 1.2681,Z 158,A -2.4301,B 24.9599,C -1.4638,E1 25.1598,E2 448.9513} C_DIS
LIN {X 136.6987,Y 5.3802,Z 158,A -0.8425,B 24.9599,C -1.4617,E1 25.1596,E2 447.3781} C_DIS
LIN {X 136.4785,Y 9.453,Z 158,A 0.8776,B 24.9596,C -1.4681,E1 25.1593,E2 445.6534} C_DIS
LIN {X 136.183,Y 13.0249,Z 158,A 2.4088,B 24.9593,C -1.4748,E1 25.1589,E2 444.1155} C_DIS
LIN {X 135.6903,Y 17.4275,Z 158,A 4.2117,B 24.9591,C -1.4778,E1 25.1583,E2 442.3161} C_DIS
LIN {X 135.1926,Y 20.938,Z 158,A 5.661,B 24.9589,C -1.4806,E1 25.1577,E2 440.8687} C_DIS
LIN {X 134.6167,Y 24.3687,Z 158,A 7.1623,B 24.9585,C -1.4878,E1 25.157,E2 439.3591} C_DIS
LIN {X 133.7667,Y 28.6691,Z 158,A 8.9968,B 24.9582,C -1.4937,E1 25.156,E2 437.5216} C_DIS
LIN {X 132.7969,Y 32.8787,Z 158,A 10.8106,B 24.9579,C -1.4996,E1 25.1548,E2 435.7043} C_DIS
LIN {X 131.8736,Y 36.4002,Z 158,A 12.2873,B 24.9578,C -1.5017,E1 25.1537,E2 434.2311} C_DIS
LIN {X 130.7759,Y 40.1629,Z 158,A 13.8395,B 24.9578,C -1.5017,E1 25.1525,E2 432.6878} C_DIS
LIN {X 129.943,Y 42.7831,Z 158,A 15.0669,B 24.9573,C -1.5096,E1 25.1514,E2 431.4487} C_DIS
LIN {X 128.0372,Y 48.186,Z 158,A 17.4118,B 24.9571,C -1.5138,E1 25.1492,E2 429.1071} C_DIS
LIN {X 126.5436,Y 51.9876,Z 158,A 19.1708,B 24.9566,C -1.5217,E1 25.1474,E2 427.3392} C_DIS
LIN {X 125.0902,Y 55.3899,Z 158,A 20.592,B 24.9568,C -1.5189,E1 25.1458,E2 425.9322} C_DIS
LIN {X 123.7327,Y 58.3612,Z 158,A 21.9447,B 24.9566,C -1.5221,E1 25.1442,E2 424.5796} C_DIS
LIN {X 122.0909,Y 61.7194,Z 158,A 23.5054,B 24.9564,C -1.5263,E1 25.1423,E2 423.0171} C_DIS
LIN {X 120.38,Y 64.9971,Z 158,A 25.1779,B 24.9557,C -1.5377,E1 25.1401,E2 421.3265} C_DIS
LIN {X 118.2847,Y 68.7362,Z 158,A 26.8986,B 24.9557,C -1.5385,E1 25.1377,E2 419.613} C_DIS
LIN {X 116.1524,Y 72.2807,Z 158,A 28.7056,B 24.9551,C -1.5475,E1 25.135,E2 417.794} C_DIS
LIN {X 114.3333,Y 75.1251,Z 158,A 30.3523,B 24.9541,C -1.5645,E1 25.1325,E2 416.1153} C_DIS
LIN {X 112.3333,Y 78.0839,Z 158,A 31.5975,B 24.9547,C -1.5541,E1 25.1305,E2 414.9007} C_DIS
LIN {X 109.7154,Y 81.7215,Z 158,A 33.4424,B 24.9546,C -1.5571,E1 25.1275,E2 413.0576} C_DIS
LIN {X 106.8777,Y 85.3996,Z 158,A 35.319,B 24.9546,C -1.558,E1 25.1243,E2 411.1878} C_DIS
LIN {X 104.1804,Y 88.6698,Z 158,A 37.1657,B 24.954,C -1.5663,E1 25.1209,E2 409.3299} C_DIS
LIN {X 101.3988,Y 91.8377,Z 158,A 38.8726,B 24.954,C -1.5672,E1 25.1178,E2 407.6286} C_DIS
LIN {X 98.704,Y 94.7284,Z 158,A 40.5707,B 24.9536,C -1.5733,E1 25.1145,E2 405.9234} C_DIS
LIN {X 95.9279,Y 97.5384,Z 158,A 42.2221,B 24.9534,C -1.5768,E1 25.1112,E2 404.2707} C_DIS
LIN {X 92.8082,Y 100.5117,Z 158,A 43.9991,B 24.9533,C -1.579,E1 25.1076,E2 402.4958} C_DIS
LIN {X 89.5373,Y 103.4362,Z 158,A 46.0409,B 24.9524,C -1.5943,E1 25.1033,E2 400.426} C_DIS
LIN {X 87.0003,Y 105.579,Z 158,A 47.1647,B 24.9531,C -1.582,E1 25.1009,E2 399.3355} C_DIS
LIN {X 83.6405,Y 108.2598,Z 158,A 48.9834,B 24.9528,C -1.5865,E1 25.0969,E2 397.5131} C_DIS
LIN {X 80.6899,Y 110.4769,Z 158,A 50.5818,B 24.9525,C -1.5922,E1 25.0933,E2 395.9068} C_DIS
LIN {X 76.9101,Y 113.1406,Z 158,A 52.4382,B 24.9525,C -1.5911,E1 25.0891,E2 394.0594} C_DIS
LIN {X 73.3952,Y 115.4522,Z 158,A 54.2715,B 24.9522,C -1.5979,E1 25.0847,E2 392.216} C_DIS
LIN {X 69.8878,Y 117.6078,Z 158,A 55.8982,B 24.9523,C -1.5951,E1 25.0809,E2 390.6009} C_DIS
LIN {X 66.3039,Y 119.6649,Z 158,A 57.6622,B 24.9521,C -1.5995,E1 25.0766,E2 388.8317} C_DIS
LIN {X 62.2747,Y 121.8082,Z 158,A 59.5097,B 24.9521,C -1.5986,E1 25.072,E2 386.9915} C_DIS
LIN {X 59.2905,Y 123.2887,Z 158,A 60.8987,B 24.9521,C -1.6,E1 25.0685,E2 385.6028} C_DIS
LIN {X 56.4018,Y 124.6376,Z 158,A 63.6699,B 24.947,C -1.6816,E1 25.0611,E2 382.6455} C_DIS
LIN {X 47.5877,Y 128.2613,Z 158,A 66.2161,B 24.9517,C -1.6052,E1 25.0549,E2 380.2857} C_DIS
LIN {X 43.73,Y 129.6277,Z 158,A 67.8666,B 24.9518,C -1.6032,E1 25.0505,E2 378.6431} C_DIS
LIN {X 40.3352,Y 130.7232,Z 158,A 69.4117,B 24.9516,C -1.6072,E1 25.0464,E2 377.0914} C_DIS
LIN {X 36.9977,Y 131.7064,Z 158,A 70.8991,B 24.9514,C -1.6099,E1 25.0424,E2 375.6001} C_DIS
LIN {X 33.4864,Y 132.6427,Z 158,A 72.3775,B 24.9515,C -1.6085,E1 25.0384,E2 374.1272} C_DIS
LIN {X 30.0581,Y 133.462,Z 158,A 73.9869,B 24.951,C -1.6166,E1 25.034,E2 372.501} C_DIS
LIN {X 26.1157,Y 134.2892,Z 158,A 75.6301,B 24.9511,C -1.615,E1 25.0295,E2 370.8637} C_DIS
LIN {X 22.1828,Y 134.9943,Z 158,A 77.3036,B 24.9511,C -1.6156,E1 25.0249,E2 369.1905} C_DIS
LIN {X 18.0585,Y 135.6076,Z 158,A 79.0222,B 24.9511,C -1.6146,E1 25.0201,E2 367.4757} C_DIS
LIN {X 14.0945,Y 136.0776,Z 158,A 80.7696,B 24.9509,C -1.6189,E1 25.0153,E2 365.7192} C_DIS
LIN {X 8.9493,Y 136.5125,Z 158,A 82.8861,B 24.951,C -1.6165,E1 25.0094,E2 363.6094} C_DIS
LIN {X 4.7431,Y 136.7236,Z 158,A 84.684,B 24.951,C -1.6182,E1 25.0044,E2 361.808} C_DIS
LIN {X 0.8378,Y 136.8021,Z 158,A 86.2006,B 24.9513,C -1.6116,E1 25.0002,E2 360.3073} C_DIS
LIN {X -3.106,Y 136.7711,Z 158,A 87.9137,B 24.9512,C -1.6145,E1 24.9954,E2 358.5873} C_DIS
LIN {X -6.7985,Y 136.6355,Z 158,A 89.4732,B 24.9512,C -1.6146,E1 24.991,E2 357.0271} C_DIS
LIN {X -11.3043,Y 136.3368,Z 158,A 91.2975,B 24.9514,C -1.6102,E1 24.986,E2 355.2125} C_DIS
LIN {X -14.7798,Y 136.0038,Z 158,A 92.7526,B 24.9514,C -1.609,E1 24.9819,E2 353.7594} C_DIS
LIN {X -18.8632,Y 135.4986,Z 158,A 94.5086,B 24.9514,C -1.6097,E1 24.9771,E2 352.0005} C_DIS
LIN {X -22.1833,Y 134.9942,Z 158,A 95.9245,B 24.9514,C -1.6092,E1 24.9731,E2 350.5846} C_DIS
LIN {X -25.7904,Y 134.3514,Z 158,A 97.4278,B 24.9517,C -1.6063,E1 24.969,E2 349.0865} C_DIS
LIN {X -29.6716,Y 133.5502,Z 158,A 99.2284,B 24.9513,C -1.6122,E1 24.9641,E2 347.2696} C_DIS
LIN {X -33.5973,Y 132.6146,Z 158,A 100.7722,B 24.9519,C -1.6029,E1 24.9599,E2 345.7457} C_DIS
LIN {X -38.2848,Y 131.3381,Z 158,A 103.1385,B 24.9509,C -1.6182,E1 24.9535,E2 343.3395} C_DIS
LIN {X -41.5583,Y 130.3391,Z 158,A 104.8563,B 24.9501,C -1.6315,E1 24.9488,E2 341.5871} C_DIS
LIN {X -46.2381,Y 128.7534,Z 158,A 106.2467,B 24.9524,C -1.5931,E1 24.9454,E2 340.2851} C_DIS
LIN {X -49.3832,Y 127.5802,Z 158,A 107.7075,B 24.9524,C -1.594,E1 24.9416,E2 338.8189} C_DIS
LIN {X -52.7395,Y 126.2295,Z 158,A 109.1242,B 24.9528,C -1.5867,E1 24.9379,E2 337.4164} C_DIS
LIN {X -55.2241,Y 125.1644,Z 158,A 110.3934,B 24.9525,C -1.5921,E1 24.9346,E2 336.1314} C_DIS
LIN {X -58.6194,Y 123.6093,Z 158,A 112.005,B 24.9525,C -1.5921,E1 24.9306,E2 334.5157} C_DIS
LIN {X -61.8119,Y 122.0439,Z 158,A 113.4017,B 24.9529,C -1.5849,E1 24.9271,E2 333.1325} C_DIS
LIN {X -65.1212,Y 120.3133,Z 158,A 115.1085,B 24.9527,C -1.5896,E1 24.9229,E2 331.4099} C_DIS
LIN {X -68.9254,Y 118.1751,Z 158,A 117.2404,B 24.9519,C -1.602,E1 24.9176,E2 329.242} C_DIS
LIN {X -72.0884,Y 116.272,Z 158,A 118.4812,B 24.953,C -1.5832,E1 24.9148,E2 328.042} C_DIS
LIN {X -75.3477,Y 114.1868,Z 158,A 120.1416,B 24.9531,C -1.5821,E1 24.9109,E2 326.3789} C_DIS
LIN {X -78.9617,Y 111.7181,Z 158,A 121.733,B 24.9541,C -1.5659,E1 24.9073,E2 324.8206} C_DIS
LIN {X -81.2163,Y 110.0903,Z 158,A 123.0619,B 24.9537,C -1.5719,E1 24.9042,E2 323.4728} C_DIS
LIN {X -84.3761,Y 107.6874,Z 158,A 124.8095,B 24.9537,C -1.5726,E1 24.9004,E2 321.7171} C_DIS
LIN {X -87.7453,Y 104.9604,Z 158,A 126.6337,B 24.9539,C -1.569,E1 24.8964,E2 319.8947} C_DIS
LIN {X -91.0009,Y 102.151,Z 158,A 128.3613,B 24.9543,C -1.561,E1 24.8928,E2 318.1792} C_DIS
LIN {X -93.5579,Y 99.8145,Z 158,A 129.9529,B 24.9541,C -1.5647,E1 24.8895,E2 316.5723} C_DIS
LIN {X -96.8615,Y 96.6116,Z 158,A 131.8491,B 24.9545,C -1.5584,E1 24.8858,E2 314.6831} C_DIS
LIN {X -99.9202,Y 93.4447,Z 158,A 133.5938,B 24.9551,C -1.5487,E1 24.8825,E2 312.9541} C_DIS
LIN {X -102.4529,Y 90.6603,Z 158,A 135.2635,B 24.9551,C -1.5493,E1 24.8793,E2 311.2753} C_DIS
LIN {X -105.1888,Y 87.4715,Z 158,A 137.058,B 24.9551,C -1.5464,E1 24.8761,E2 309.4796} C_DIS
LIN {X -107.7643,Y 84.2782,Z 158,A 138.7107,B 24.9557,C -1.5384,E1 24.8732,E2 307.8381} C_DIS
LIN {X -113.3291,Y 76.6316,Z 158,A 142.5728,B 24.9566,C -1.5222,E1 24.867,E2 303.996} C_DIS
LIN {X -115.1047,Y 73.9379,Z 158,A 144.1506,B 24.9562,C -1.5297,E1 24.8645,E2 302.3922} C_DIS
LIN {X -117.6307,Y 69.8494,Z 158,A 146.1693,B 24.9565,C -1.5241,E1 24.8616,E2 300.3765} C_DIS
LIN {X -119.9365,Y 65.8121,Z 158,A 148.038,B 24.957,C -1.5143,E1 24.8591,E2 298.5213} C_DIS
LIN {X -121.7687,Y 62.3525,Z 158,A 149.6904,B 24.9573,C -1.51,E1 24.857,E2 296.8704} C_DIS
LIN {X -123.2197,Y 59.435,Z 158,A 150.9522,B 24.9578,C -1.5006,E1 24.8554,E2 295.624} C_DIS
LIN {X -124.7333,Y 56.1879,Z 158,A 152.5596,B 24.9578,C -1.5014,E1 24.8535,E2 294.0061} C_DIS
LIN {X -126.0081,Y 53.2698,Z 158,A 153.8674,B 24.9581,C -1.4959,E1 24.8521,E2 292.7041} C_DIS
Enddeposition()
END
